KUKA KRL program: MyProgram_064().src

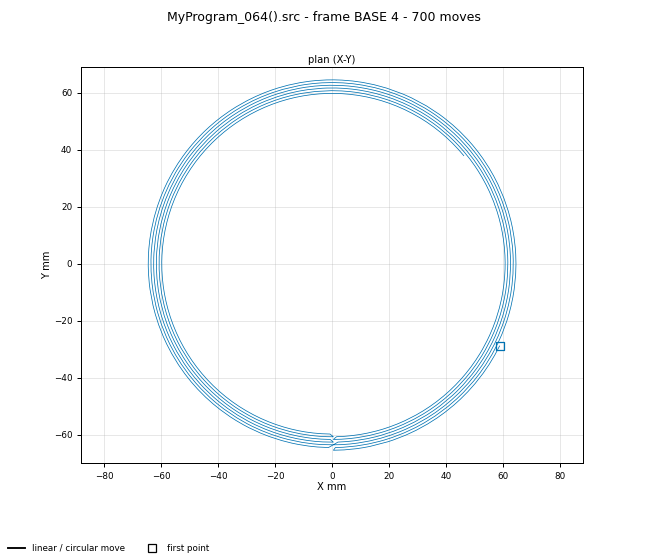
[picture p0: tool path of MyProgram_064().src in frame BASE 4, 700 of 700 moves have a stored position in this frame; points joined in program order, loops and branches not executed]
&ACCESS RVP
&REL 1
&PARAM TEMPLATE = C:\KRC\Roboter\Template\vorgabe
&PARAM EDITMASK = *
DEF MyProgram_064()
; ---- Setting reference (Base) ----
$BASE = BASE_DATA[4]

; --------------------------
; ---- Setting tool (TCP) ----
$TOOL = TOOL_DATA[3]
; --------------------------

$VEL.CP = VEL_APROX_PRINT
Startdeposition()
$VEL.CP = VEL_PRINT
LIN {X 58.7468,Y -28.8662,Z 73,A -33.1433,B 24.8941,C -2.3753,E1 25.1418,E2 117.3384} C_DIS
LIN {X 57.128,Y -31.9497,Z 73,A -36.5438,B 24.8957,C -2.3576,E1 25.1372,E2 120.763} C_DIS
LIN {X 55.082,Y -35.3604,Z 73,A -38.4998,B 24.8931,C -2.3868,E1 25.1344,E2 122.6401} C_DIS
LIN {X 52.9744,Y -38.4471,Z 73,A -42.3446,B 24.8952,C -2.3631,E1 25.1282,E2 126.522} C_DIS
LIN {X 50.1872,Y -42.0184,Z 73,A -46.4103,B 24.8964,C -2.3503,E1 25.1211,E2 130.5991} C_DIS
LIN {X 47.6348,Y -44.8923,Z 73,A -49.7399,B 24.897,C -2.3428,E1 25.1148,E2 133.9318} C_DIS
LIN {X 44.9577,Y -47.5733,Z 73,A -52.5816,B 24.8967,C -2.3469,E1 25.1092,E2 136.7518} C_DIS
LIN {X 42.7353,Y -49.5785,Z 73,A -55.4715,B 24.8978,C -2.3342,E1 25.1031,E2 139.6603} C_DIS
LIN {X 39.675,Y -52.0599,Z 73,A -59.4462,B 24.8996,C -2.3137,E1 25.0943,E2 143.6687} C_DIS
LIN {X 36.8552,Y -54.0936,Z 73,A -62.9268,B 24.901,C -2.297,E1 25.0862,E2 147.1772} C_DIS
LIN {X 33.4783,Y -56.2461,Z 73,A -64.9571,B 24.8984,C -2.3268,E1 25.0815,E2 149.1305} C_DIS
LIN {X 29.5121,Y -58.4253,Z 73,A -69.386,B 24.9,C -2.3085,E1 25.0706,E2 153.5901} C_DIS
LIN {X 25.8118,Y -60.1522,Z 73,A -72.5953,B 24.8997,C -2.3119,E1 25.0625,E2 156.7831} C_DIS
LIN {X 21.4205,Y -61.8516,Z 73,A -76.9276,B 24.9006,C -2.3013,E1 25.0511,E2 161.1313} C_DIS
LIN {X 19.5492,Y -62.468,Z 73,A -79.1991,B 24.9019,C -2.2862,E1 25.045,E2 163.4345} C_DIS
LIN {X 13.289,Y -64.0922,Z 73,A -83.8581,B 24.9004,C -2.3046,E1 25.0325,E2 168.0431} C_DIS
LIN {X 10.9976,Y -64.5247,Z 73,A -86.2924,B 24.9013,C -2.2936,E1 25.0257,E2 170.5007} C_DIS
LIN {X 8.6432,Y -64.8825,Z 73,A -88.6806,B 24.902,C -2.2851,E1 25.0191,E2 172.9071} C_DIS
LIN {X 4.2204,Y -65.3193,Z 73,A -92.8829,B 24.9028,C -2.2759,E1 25.0073,E2 177.1288} C_DIS
LIN {X 0.4624,Y -65.4389,Z 73,A -95.428,B 24.9014,C -2.2924,E1 25.0003,E2 179.6343} C_DIS
Enddeposition()
LIN {X 0.4624,Y -65.4389,Z 73,A -95.428,B 24.9014,C -2.2924,E1 25.0003,E2 179.6343} C_DIS
Startdeposition()
$VEL.CP = VEL_PRINT
LIN {X 1.1563,Y -64.495,Z 73,A -93.473,B 24.8973,C -2.3399,E1 25.0061,E2 177.5667} C_DIS
LIN {X 3.9215,Y -64.387,Z 73,A -91.3651,B 24.8979,C -2.3327,E1 25.0119,E2 175.4769} C_DIS
LIN {X 8.4282,Y -63.9525,Z 73,A -87.3099,B 24.8976,C -2.3358,E1 25.0232,E2 171.4172} C_DIS
LIN {X 12.7281,Y -63.2376,Z 73,A -83.9125,B 24.8984,C -2.3275,E1 25.0325,E2 168.0431} C_DIS
LIN {X 16.6215,Y -62.3274,Z 73,A -80.4027,B 24.8982,C -2.3299,E1 25.042,E2 164.5326} C_DIS
LIN {X 18.4457,Y -61.8118,Z 73,A -78.1953,B 24.8969,C -2.3443,E1 25.048,E2 162.2946} C_DIS
LIN {X 21.0877,Y -60.9617,Z 73,A -75.1268,B 24.8953,C -2.3621,E1 25.0562,E2 159.1901} C_DIS
LIN {X 25.2751,Y -59.3478,Z 73,A -71.5296,B 24.8957,C -2.3581,E1 25.0655,E2 155.6106} C_DIS
LIN {X 29.3295,Y -57.4519,Z 73,A -67.1057,B 24.8941,C -2.3757,E1 25.0766,E2 151.157} C_DIS
LIN {X 32.259,Y -55.8598,Z 73,A -65.0308,B 24.8956,C -2.3588,E1 25.0815,E2 149.1282} C_DIS
LIN {X 36.0916,Y -53.4634,Z 73,A -60.9163,B 24.8947,C -2.3688,E1 25.0912,E2 145.0033} C_DIS
LIN {X 40.6403,Y -50.093,Z 73,A -55.6203,B 24.8932,C -2.3861,E1 25.103,E2 139.6857} C_DIS
LIN {X 43.7386,Y -47.4121,Z 73,A -52.4535,B 24.8935,C -2.3824,E1 25.1096,E2 136.5403} C_DIS
LIN {X 46.088,Y -45.1316,Z 73,A -48.8099,B 24.8912,C -2.4081,E1 25.1169,E2 132.8512} C_DIS
LIN {X 49.6452,Y -41.1861,Z 73,A -44.3491,B 24.8907,C -2.4135,E1 25.125,E2 128.398} C_DIS
LIN {X 51.7521,Y -38.5064,Z 73,A -40.8175,B 24.8888,C -2.4346,E1 25.131,E2 124.8333} C_DIS
LIN {X 53.8109,Y -35.5715,Z 73,A -38.7033,B 24.8905,C -2.4156,E1 25.1342,E2 122.7745} C_DIS
LIN {X 56.1541,Y -31.7454,Z 73,A -34.9176,B 24.8899,C -2.4217,E1 25.1396,E2 118.9938} C_DIS
LIN {X 58.1359,Y -27.949,Z 73,A -31.0519,B 24.8888,C -2.4344,E1 25.1446,E2 115.1186} C_DIS
LIN {X 59.5801,Y -24.7239,Z 73,A -27.7511,B 24.8875,C -2.4479,E1 25.1483,E2 111.8037} C_DIS
LIN {X 61.2868,Y -20.1226,Z 73,A -23.7571,B 24.8872,C -2.4517,E1 25.1521,E2 107.8231} C_DIS
LIN {X 62.0906,Y -17.4843,Z 73,A -20.6908,B 24.885,C -2.4754,E1 25.1545,E2 104.7185} C_DIS
LIN {X 62.7454,Y -14.9688,Z 73,A -17.8709,B 24.8831,C -2.496,E1 25.1564,E2 101.8661} C_DIS
LIN {X 63.4244,Y -11.762,Z 73,A -15.9567,B 24.8847,C -2.479,E1 25.1573,E2 100.0033} C_DIS
LIN {X 63.8772,Y -8.9808,Z 73,A -12.9667,B 24.8827,C -2.4997,E1 25.1586,E2 96.982} C_DIS
LIN {X 64.3886,Y -3.8939,Z 73,A -8.1546,B 24.8807,C -2.5212,E1 25.1597,E2 92.1478} C_DIS
LIN {X 64.5052,Y -0.0652,Z 73,A -4.5358,B 24.8791,C -2.5377,E1 25.1597,E2 88.5115} C_DIS
LIN {X 64.4157,Y 3.4022,Z 73,A -2.7198,B 24.8813,C -2.5142,E1 25.1595,E2 86.7617} C_DIS
LIN {X 64.2639,Y 5.5868,Z 73,A -0.0027,B 24.8788,C -2.5404,E1 25.1589,E2 83.9987} C_DIS
LIN {X 63.8203,Y 9.3812,Z 73,A 3.0196,B 24.8788,C -2.5413,E1 25.1578,E2 80.9922} C_DIS
LIN {X 63.2661,Y 12.5892,Z 73,A 5.7276,B 24.8784,C -2.5454,E1 25.1564,E2 78.2903} C_DIS
LIN {X 62.7327,Y 15.0207,Z 73,A 8.8882,B 24.8753,C -2.5769,E1 25.1544,E2 75.0737} C_DIS
LIN {X 61.8474,Y 18.326,Z 73,A 11.5961,B 24.8753,C -2.5773,E1 25.1522,E2 72.3804} C_DIS
LIN {X 60.2454,Y 23.0538,Z 73,A 15.908,B 24.8744,C -2.5869,E1 25.1481,E2 68.0698} C_DIS
LIN {X 58.1702,Y 27.8777,Z 73,A 19.5732,B 24.8756,C -2.5744,E1 25.1441,E2 64.4542} C_DIS
LIN {X 56.6801,Y 30.7946,Z 73,A 23.2418,B 24.8729,C -2.6016,E1 25.1393,E2 60.7406} C_DIS
LIN {X 55.1029,Y 33.5352,Z 73,A 25.9438,B 24.8725,C -2.6062,E1 25.1354,E2 58.0416} C_DIS
LIN {X 52.9089,Y 36.8998,Z 73,A 29.262,B 24.8722,C -2.6088,E1 25.1303,E2 54.7336} C_DIS
LIN {X 51.0307,Y 39.4563,Z 73,A 32.2683,B 24.8711,C -2.6204,E1 25.1252,E2 51.7143} C_DIS
LIN {X 49.2652,Y 41.6406,Z 73,A 34.9272,B 24.8701,C -2.6302,E1 25.1204,E2 49.0442} C_DIS
LIN {X 47.4786,Y 43.666,Z 73,A 37.4243,B 24.8693,C -2.638,E1 25.1157,E2 46.5399} C_DIS
LIN {X 44.7609,Y 46.4478,Z 73,A 41.2384,B 24.8677,C -2.6541,E1 25.108,E2 42.7035} C_DIS
LIN {X 42.3154,Y 48.6864,Z 73,A 42.8652,B 24.8704,C -2.6272,E1 25.1048,E2 41.147} C_DIS
LIN {X 39.4678,Y 51.022,Z 73,A 46.1417,B 24.8698,C -2.6333,E1 25.0977,E2 37.8684} C_DIS
LIN {X 37.6241,Y 52.3966,Z 73,A 49.0641,B 24.8673,C -2.6583,E1 25.091,E2 34.8972} C_DIS
LIN {X 33.1232,Y 55.3526,Z 73,A 54.1357,B 24.8659,C -2.6725,E1 25.079,E2 29.8081} C_DIS
LIN {X 27.7921,Y 58.2114,Z 73,A 58.8294,B 24.8668,C -2.6629,E1 25.0674,E2 25.15} C_DIS
LIN {X 24.9466,Y 59.486,Z 73,A 62.2777,B 24.8649,C -2.6821,E1 25.0584,E2 21.6645} C_DIS
LIN {X 19.1378,Y 61.601,Z 73,A 67.412,B 24.8653,C -2.6781,E1 25.0449,E2 16.5496} C_DIS
LIN {X 14.7147,Y 62.8049,Z 73,A 71.1148,B 24.8659,C -2.672,E1 25.035,E2 12.8672} C_DIS
LIN {X 10.6426,Y 63.6213,Z 73,A 74.7482,B 24.8659,C -2.6721,E1 25.025,E2 9.2375} C_DIS
LIN {X 7.1714,Y 64.1051,Z 73,A 78.0569,B 24.8654,C -2.6772,E1 25.0158,E2 5.9193} C_DIS
LIN {X 3.4827,Y 64.4113,Z 73,A 81.5905,B 24.8648,C -2.6829,E1 25.0059,E2 2.3739} C_DIS
LIN {X 0.7153,Y 64.5022,Z 73,A 83.698,B 24.8657,C -2.6746,E1 25.0001,E2 0.2864} C_DIS
LIN {X -1.9461,Y 64.476,Z 73,A 86.182,B 24.8655,C -2.6766,E1 24.9932,E2 -2.2028} C_DIS
LIN {X -5.6035,Y 64.2621,Z 73,A 89.1745,B 24.8662,C -2.6695,E1 24.9849,E2 -5.1793} C_DIS
LIN {X -7.8512,Y 64.0265,Z 73,A 91.6622,B 24.8652,C -2.6789,E1 24.9779,E2 -7.6912} C_DIS
LIN {X -11.169,Y 63.5315,Z 73,A 93.8899,B 24.8671,C -2.6604,E1 24.9719,E2 -9.8769} C_DIS
LIN {X -15.3244,Y 62.6586,Z 73,A 97.4252,B 24.8679,C -2.6521,E1 24.9623,E2 -13.3967} C_DIS
LIN {X -18.975,Y 61.6515,Z 73,A 101.1903,B 24.8674,C -2.6572,E1 24.9521,E2 -17.1798} C_DIS
LIN {X -21.3436,Y 60.8719,Z 73,A 103.7868,B 24.8669,C -2.6626,E1 24.9452,E2 -19.7943} C_DIS
LIN {X -23.8319,Y 59.9421,Z 73,A 105.8647,B 24.8678,C -2.6535,E1 24.9398,E2 -21.8549} C_DIS
LIN {X -26.8305,Y 58.6604,Z 73,A 109.1217,B 24.8674,C -2.6569,E1 24.9314,E2 -25.1278} C_DIS
LIN {X -29.8299,Y 57.1928,Z 73,A 112.1913,B 24.8677,C -2.6544,E1 24.9238,E2 -28.1996} C_DIS
LIN {X -33.6214,Y 55.0505,Z 73,A 116.1114,B 24.8683,C -2.6486,E1 24.9144,E2 -32.1176} C_DIS
LIN {X -35.7625,Y 53.6849,Z 73,A 118.4897,B 24.8685,C -2.6468,E1 24.9088,E2 -34.4995} C_DIS
LIN {X -38.7189,Y 51.5925,Z 73,A 121.1599,B 24.8702,C -2.6291,E1 24.9029,E2 -37.1368} C_DIS
LIN {X -40.7762,Y 49.9828,Z 73,A 123.624,B 24.8704,C -2.6271,E1 24.8975,E2 -39.6053} C_DIS
LIN {X -43.021,Y 48.0638,Z 73,A 126.3383,B 24.8708,C -2.6231,E1 24.8918,E2 -42.3208} C_DIS
LIN {X -44.9132,Y 46.301,Z 73,A 128.3455,B 24.8719,C -2.6119,E1 24.8878,E2 -44.3096} C_DIS
LIN {X -47.0355,Y 44.143,Z 73,A 131.0757,B 24.8725,C -2.6062,E1 24.8825,E2 -47.0381} C_DIS
LIN {X -49.1146,Y 41.8173,Z 73,A 134.0295,B 24.8728,C -2.603,E1 24.877,E2 -49.9973} C_DIS
LIN {X -50.8555,Y 39.682,Z 73,A 136.4233,B 24.8735,C -2.5956,E1 24.8729,E2 -52.3846} C_DIS
LIN {X -52.3173,Y 37.7353,Z 73,A 139.0436,B 24.8732,C -2.5989,E1 24.8685,E2 -55.0256} C_DIS
LIN {X -54.1138,Y 35.1103,Z 73,A 141.9232,B 24.8738,C -2.5922,E1 24.8641,E2 -57.9037} C_DIS
LIN {X -56.0657,Y 31.9007,Z 73,A 145.8862,B 24.8735,C -2.5953,E1 24.8585,E2 -61.8947} C_DIS
LIN {X -57.8264,Y 28.584,Z 73,A 147.8932,B 24.877,C -2.5593,E1 24.8561,E2 -63.8264} C_DIS
LIN {X -58.8491,Y 26.4142,Z 73,A 150.8405,B 24.8761,C -2.569,E1 24.8526,E2 -66.8131} C_DIS
LIN {X -60.0746,Y 23.4945,Z 73,A 153.3783,B 24.8774,C -2.5551,E1 24.85,E2 -69.3319} C_DIS
LIN {X -61.2817,Y 20.139,Z 73,A 156.0607,B 24.8793,C -2.536,E1 24.8476,E2 -71.9838} C_DIS
LIN {X -62.395,Y 16.3677,Z 73,A 159.7267,B 24.88,C -2.5285,E1 24.8448,E2 -75.6532} C_DIS
LIN {X -63.4409,Y 11.673,Z 73,A 164.467,B 24.8804,C -2.5242,E1 24.842,E2 -80.4111} C_DIS
LIN {X -63.9424,Y 8.506,Z 73,A 167.1894,B 24.8815,C -2.5128,E1 24.8409,E2 -83.1225} C_DIS
LIN {X -64.2894,Y 5.2748,Z 73,A 169.9321,B 24.8826,C -2.5009,E1 24.8402,E2 -85.8531} C_DIS
LIN {X -64.4537,Y 2.5868,Z 73,A 172.7814,B 24.8825,C -2.5022,E1 24.8398,E2 -88.7227} C_DIS
LIN {X -64.5026,Y -0.6904,Z 73,A 175.1299,B 24.8844,C -2.482,E1 24.8398,E2 -91.0371} C_DIS
LIN {X -64.4131,Y -3.4495,Z 73,A 177.9855,B 24.8844,C -2.4822,E1 24.8402,E2 -93.9102} C_DIS
LIN {X -64.1273,Y -6.9783,Z 73,A -179.2847,B 24.886,C -2.4642,E1 24.8408,E2 -96.6136} C_DIS
LIN {X -63.8745,Y -8.9997,Z 73,A -177.1157,B 24.8859,C -2.4657,E1 24.8417,E2 -98.7989} C_DIS
LIN {X -62.8104,Y -14.6909,Z 73,A -172.4745,B 24.8883,C -2.4401,E1 24.8441,E2 -103.4064} C_DIS
LIN {X -61.9956,Y -17.8198,Z 73,A -168.0907,B 24.8863,C -2.4614,E1 24.8475,E2 -107.8666} C_DIS
LIN {X -60.8295,Y -21.4645,Z 73,A -165.918,B 24.8895,C -2.427,E1 24.8494,E2 -109.9696} C_DIS
LIN {X -59.2781,Y -25.4398,Z 73,A -161.8551,B 24.8899,C -2.4216,E1 24.8536,E2 -114.0421} C_DIS
LIN {X -58.0145,Y -28.2019,Z 73,A -158.1558,B 24.8888,C -2.4344,E1 24.8581,E2 -117.792} C_DIS
LIN {X -56.2629,Y -31.5505,Z 73,A -155.8796,B 24.8916,C -2.4035,E1 24.8611,E2 -120.0065} C_DIS
LIN {X -53.8835,Y -35.4614,Z 73,A -152.2506,B 24.8933,C -2.3842,E1 24.8664,E2 -123.6081} C_DIS
LIN {X -51.6586,Y -38.6308,Z 73,A -148.4743,B 24.8935,C -2.3826,E1 24.8725,E2 -127.3988} C_DIS
LIN {X -49.5171,Y -41.3402,Z 73,A -144.8664,B 24.8931,C -2.3865,E1 24.8789,E2 -131.033} C_DIS
LIN {X -47.1087,Y -44.0652,Z 73,A -141.5659,B 24.8936,C -2.3809,E1 24.8851,E2 -134.3347} C_DIS
LIN {X -44.345,Y -46.8455,Z 73,A -138.75,B 24.8955,C -2.3599,E1 24.8906,E2 -137.1124} C_DIS
LIN {X -41.6698,Y -49.2404,Z 73,A -135.7027,B 24.8963,C -2.3508,E1 24.897,E2 -140.15} C_DIS
LIN {X -39.2021,Y -51.2263,Z 73,A -132.6426,B 24.8963,C -2.3508,E1 24.9037,E2 -143.2217} C_DIS
LIN {X -35.7236,Y -53.7106,Z 73,A -128.9483,B 24.897,C -2.3424,E1 24.9121,E2 -146.9086} C_DIS
LIN {X -33.6688,Y -55.0217,Z 73,A -126.382,B 24.8966,C -2.3477,E1 24.9182,E2 -149.4957} C_DIS
LIN {X -31.0087,Y -56.5632,Z 73,A -123.8018,B 24.8972,C -2.3408,E1 24.9245,E2 -152.0669} C_DIS
LIN {X -29.1203,Y -57.5588,Z 73,A -121.5169,B 24.8967,C -2.3468,E1 24.9302,E2 -154.3723} C_DIS
LIN {X -25.066,Y -59.436,Z 73,A -117.0106,B 24.896,C -2.3545,E1 24.9418,E2 -158.9076} C_DIS
LIN {X -22.0591,Y -60.6163,Z 73,A -114.5932,B 24.8971,C -2.3419,E1 24.9481,E2 -161.3} C_DIS
LIN {X -17.6643,Y -62.0396,Z 73,A -110.5991,B 24.8976,C -2.3365,E1 24.9587,E2 -165.2882} C_DIS
LIN {X -14.1336,Y -62.9391,Z 73,A -107.5975,B 24.8982,C -2.3296,E1 24.9668,E2 -168.2773} C_DIS
LIN {X -11.91,Y -63.3958,Z 73,A -104.5581,B 24.8962,C -2.3522,E1 24.9753,E2 -171.3737} C_DIS
LIN {X -8.2112,Y -63.9806,Z 73,A -102.147,B 24.8981,C -2.3305,E1 24.9819,E2 -173.7351} C_DIS
LIN {X -5.2225,Y -64.2936,Z 73,A -99.2022,B 24.8976,C -2.3367,E1 24.9901,E2 -176.696} C_DIS
LIN {X -1.2767,Y -64.4928,Z 73,A -95.5948,B 24.8973,C -2.3394,E1 25.0002,E2 -180.3105} C_DIS
LIN {X -1.2767,Y -64.4928,Z 73,A -95.5948,B 24.8973,C -2.3394,E1 25.0002,E2 -180.3105} C_DIS
Enddeposition()
LIN {X 0.4502,Y -63.526,Z 73,A -94.7693,B 24.8973,C -2.3401,E1 25.0025,E2 -181.1376} C_DIS
Startdeposition()
$VEL.CP = VEL_PRINT
LIN {X -3.7985,Y -63.4425,Z 73,A -99.6016,B 24.8993,C -2.3166,E1 24.9888,E2 -176.2488} C_DIS
LIN {X -6.7271,Y -63.1985,Z 73,A -102.2235,B 24.8993,C -2.3174,E1 24.9815,E2 -173.6275} C_DIS
LIN {X -10.6276,Y -62.6607,Z 73,A -106.2689,B 24.9001,C -2.3076,E1 24.9703,E2 -169.5551} C_DIS
LIN {X -15.5509,Y -61.6242,Z 73,A -110.2262,B 24.8988,C -2.3222,E1 24.9596,E2 -165.6275} C_DIS
LIN {X -17.8908,Y -60.9853,Z 73,A -112.694,B 24.8992,C -2.3176,E1 24.9529,E2 -163.1449} C_DIS
LIN {X -21.2948,Y -59.8823,Z 73,A -116.714,B 24.9004,C -2.3036,E1 24.9422,E2 -159.0836} C_DIS
LIN {X -24.7528,Y -58.5371,Z 73,A -118.827,B 24.8979,C -2.3326,E1 24.937,E2 -157.0351} C_DIS
LIN {X -27.9356,Y -57.0876,Z 73,A -122.2592,B 24.8981,C -2.3303,E1 24.9282,E2 -153.5889} C_DIS
LIN {X -29.8114,Y -56.1304,Z 73,A -124.2589,B 24.8981,C -2.3307,E1 24.9233,E2 -151.5843} C_DIS
LIN {X -33.4,Y -54.0725,Z 73,A -128.1266,B 24.8979,C -2.3331,E1 24.914,E2 -147.7107} C_DIS
LIN {X -37.9663,Y -50.9698,Z 73,A -132.4905,B 24.8961,C -2.3537,E1 24.904,E2 -143.381} C_DIS
LIN {X -40.6133,Y -48.8861,Z 73,A -135.4758,B 24.8955,C -2.3601,E1 24.8975,E2 -140.4002} C_DIS
LIN {X -42.7747,Y -47.0067,Z 73,A -138.4364,B 24.8957,C -2.3575,E1 24.8913,E2 -137.4215} C_DIS
LIN {X -45.9463,Y -43.9124,Z 73,A -142.262,B 24.8947,C -2.3691,E1 24.8837,E2 -133.6074} C_DIS
LIN {X -47.8059,Y -41.8796,Z 73,A -145.1896,B 24.895,C -2.3658,E1 24.8782,E2 -130.6589} C_DIS
LIN {X -50.2885,Y -38.8635,Z 73,A -148.4282,B 24.8937,C -2.3795,E1 24.8726,E2 -127.4379} C_DIS
LIN {X -52.8793,Y -35.2587,Z 73,A -152.507,B 24.893,C -2.3878,E1 24.866,E2 -123.359} C_DIS
LIN {X -54.9846,Y -31.8755,Z 73,A -156.0304,B 24.892,C -2.3985,E1 24.8609,E2 -119.8429} C_DIS
LIN {X -56.8065,Y -28.5003,Z 73,A -159.7696,B 24.8917,C -2.4024,E1 24.856,E2 -116.0932} C_DIS
LIN {X -58.1144,Y -25.7321,Z 73,A -162.3869,B 24.8908,C -2.4128,E1 24.853,E2 -113.4863} C_DIS
LIN {X -59.8691,Y -21.3326,Z 73,A -166.725,B 24.8898,C -2.4237,E1 24.8486,E2 -109.15} C_DIS
LIN {X -61.2709,Y -16.8902,Z 73,A -171.0555,B 24.8888,C -2.4337,E1 24.8451,E2 -104.8184} C_DIS
LIN {X -61.7704,Y -14.9572,Z 73,A -173.4635,B 24.8894,C -2.4278,E1 24.8435,E2 -102.3821} C_DIS
LIN {X -62.7382,Y -10.163,Z 73,A -177.4879,B 24.8875,C -2.4484,E1 24.8415,E2 -98.3834} C_DIS
LIN {X -63.195,Y -6.7605,Z 73,A 179.7094,B 24.8861,C -2.4635,E1 24.8405,E2 -95.6} C_DIS
LIN {X -63.4977,Y -2.7039,Z 73,A 175.8031,B 24.8854,C -2.4706,E1 24.8399,E2 -91.687} C_DIS
LIN {X -63.5426,Y 1.2841,Z 73,A 172.2845,B 24.8842,C -2.4834,E1 24.8399,E2 -88.1778} C_DIS
LIN {X -63.4473,Y 3.7097,Z 73,A 170.3781,B 24.8831,C -2.4955,E1 24.8401,E2 -86.289} C_DIS
LIN {X -63.2082,Y 6.6348,Z 73,A 167.1731,B 24.8833,C -2.4935,E1 24.8409,E2 -83.0599} C_DIS
LIN {X -62.8176,Y 9.6561,Z 73,A 164.8611,B 24.8817,C -2.5103,E1 24.8418,E2 -80.7741} C_DIS
LIN {X -62.4549,Y 11.7785,Z 73,A 162.8495,B 24.8813,C -2.515,E1 24.8428,E2 -78.7621} C_DIS
LIN {X -61.624,Y 15.5515,Z 73,A 159.5903,B 24.8798,C -2.5301,E1 24.8448,E2 -75.5197} C_DIS
LIN {X -60.4183,Y 19.7217,Z 73,A 154.7618,B 24.8803,C -2.5251,E1 24.8488,E2 -70.6515} C_DIS
LIN {X -58.8753,Y 23.9373,Z 73,A 150.0331,B 24.8803,C -2.5248,E1 24.8537,E2 -65.8955} C_DIS
LIN {X -57.1956,Y 27.7128,Z 73,A 147.753,B 24.8767,C -2.5626,E1 24.8563,E2 -63.6934} C_DIS
LIN {X -54.973,Y 31.8957,Z 73,A 143.4451,B 24.8756,C -2.5741,E1 24.862,E2 -59.3902} C_DIS
LIN {X -53.9031,Y 33.6712,Z 73,A 140.8478,B 24.8764,C -2.5656,E1 24.8658,E2 -56.7593} C_DIS
LIN {X -51.6543,Y 37.029,Z 73,A 137.545,B 24.8748,C -2.5819,E1 24.871,E2 -53.4791} C_DIS
LIN {X -49.8108,Y 39.4738,Z 73,A 135.0334,B 24.8737,C -2.5939,E1 24.8753,E2 -50.9843} C_DIS
LIN {X -48.454,Y 41.1281,Z 73,A 132.3496,B 24.8746,C -2.5844,E1 24.8802,E2 -48.2655} C_DIS
LIN {X -44.9681,Y 44.9142,Z 73,A 128.2243,B 24.8725,C -2.6055,E1 24.888,E2 -44.1726} C_DIS
LIN {X -43.0497,Y 46.7549,Z 73,A 125.9285,B 24.8718,C -2.613,E1 24.8927,E2 -41.8853} C_DIS
LIN {X -41.1909,Y 48.4004,Z 73,A 123.729,B 24.8712,C -2.6187,E1 24.8973,E2 -39.6908} C_DIS
LIN {X -39.4304,Y 49.8451,Z 73,A 121.4963,B 24.8712,C -2.6196,E1 24.9022,E2 -37.4519} C_DIS
LIN {X -37.1121,Y 51.595,Z 73,A 118.6635,B 24.871,C -2.6207,E1 24.9086,E2 -34.6116} C_DIS
LIN {X -34.0821,Y 53.6451,Z 73,A 115.5229,B 24.8701,C -2.6301,E1 24.9159,E2 -31.4831} C_DIS
LIN {X -31.4466,Y 55.2311,Z 73,A 112.4741,B 24.8701,C -2.6295,E1 24.9233,E2 -28.4237} C_DIS
LIN {X -27.9052,Y 57.1027,Z 73,A 109.1629,B 24.869,C -2.6413,E1 24.9314,E2 -25.1317} C_DIS
LIN {X -24.7861,Y 58.5231,Z 73,A 106.1589,B 24.8684,C -2.6475,E1 24.9391,E2 -22.1354} C_DIS
LIN {X -21.0077,Y 59.9831,Z 73,A 102.3305,B 24.8683,C -2.6486,E1 24.9491,E2 -18.3018} C_DIS
LIN {X -17.264,Y 61.1658,Z 73,A 98.5447,B 24.8683,C -2.6475,E1 24.9593,E2 -14.5068} C_DIS
LIN {X -11.2802,Y 62.5464,Z 73,A 93.8654,B 24.8661,C -2.6702,E1 24.9719,E2 -9.8757} C_DIS
LIN {X -9.3924,Y 62.8576,Z 73,A 91.5957,B 24.8671,C -2.6599,E1 24.9782,E2 -7.5794} C_DIS
LIN {X -6.4948,Y 63.2228,Z 73,A 88.8376,B 24.8673,C -2.6587,E1 24.9859,E2 -4.8167} C_DIS
LIN {X -3.5543,Y 63.456,Z 73,A 86.2786,B 24.8669,C -2.6619,E1 24.993,E2 -2.2644} C_DIS
LIN {X 0.1727,Y 63.5556,Z 73,A 82.8264,B 24.8671,C -2.6608,E1 25.0026,E2 1.1907} C_DIS
LIN {X 3.8336,Y 63.4394,Z 73,A 79.4792,B 24.8671,C -2.66,E1 25.012,E2 4.5388} C_DIS
LIN {X 7.4768,Y 63.1142,Z 73,A 75.8987,B 24.8678,C -2.6534,E1 25.0219,E2 8.1326} C_DIS
LIN {X 10.6917,Y 62.65,Z 73,A 72.9261,B 24.868,C -2.6514,E1 25.0301,E2 11.1068} C_DIS
LIN {X 14.9359,Y 61.7756,Z 73,A 69.3195,B 24.8675,C -2.6562,E1 25.0399,E2 14.6974} C_DIS
LIN {X 18.3372,Y 60.8532,Z 73,A 65.3416,B 24.8695,C -2.6361,E1 25.0507,E2 18.7161} C_DIS
LIN {X 21.7721,Y 59.7099,Z 73,A 63.0845,B 24.8675,C -2.6559,E1 25.0565,E2 20.9216} C_DIS
LIN {X 25.2997,Y 58.3029,Z 73,A 59.5839,B 24.8681,C -2.6506,E1 25.0655,E2 24.4266} C_DIS
LIN {X 27.9916,Y 57.0599,Z 73,A 56.4298,B 24.8695,C -2.6364,E1 25.0735,E2 27.6061} C_DIS
LIN {X 32.6289,Y 54.5414,Z 73,A 52.5017,B 24.8682,C -2.6491,E1 25.083,E2 31.4926} C_DIS
LIN {X 34.4548,Y 53.4058,Z 73,A 50.395,B 24.8689,C -2.6422,E1 25.088,E2 33.6088} C_DIS
LIN {X 36.2153,Y 52.2279,Z 73,A 47.9023,B 24.8706,C -2.6255,E1 25.0938,E2 36.1328} C_DIS
LIN {X 38.8111,Y 50.3288,Z 73,A 44.8216,B 24.8715,C -2.6161,E1 25.1007,E2 39.2243} C_DIS
LIN {X 41.5761,Y 48.0709,Z 73,A 42.3802,B 24.8703,C -2.6284,E1 25.1058,E2 41.6272} C_DIS
LIN {X 44.281,Y 45.5911,Z 73,A 39.2645,B 24.8705,C -2.6264,E1 25.1122,E2 44.735} C_DIS
LIN {X 46.1792,Y 43.667,Z 73,A 36.8142,B 24.871,C -2.6209,E1 25.1169,E2 47.1879} C_DIS
LIN {X 48.1461,Y 41.4894,Z 73,A 33.8897,B 24.8723,C -2.6082,E1 25.1224,E2 50.1292} C_DIS
LIN {X 50.8543,Y 38.1199,Z 73,A 30.2544,B 24.8726,C -2.6054,E1 25.1287,E2 53.7541} C_DIS
LIN {X 51.8988,Y 36.6863,Z 73,A 28.0406,B 24.8744,C -2.5865,E1 25.1323,E2 56.0019} C_DIS
LIN {X 53.6234,Y 34.1158,Z 73,A 25.3869,B 24.8748,C -2.5827,E1 25.1363,E2 58.6512} C_DIS
LIN {X 55.5762,Y 30.832,Z 73,A 21.9153,B 24.8757,C -2.5729,E1 25.1411,E2 62.1279} C_DIS
LIN {X 57.3051,Y 27.4849,Z 73,A 18.8513,B 24.8758,C -2.5718,E1 25.1449,E2 65.1782} C_DIS
LIN {X 58.6645,Y 24.4506,Z 73,A 15.7975,B 24.8768,C -2.562,E1 25.1483,E2 68.2386} C_DIS
LIN {X 59.6866,Y 21.8358,Z 73,A 13.2718,B 24.8775,C -2.5548,E1 25.1508,E2 70.7672} C_DIS
LIN {X 60.9388,Y 18.0486,Z 73,A 9.2871,B 24.8794,C -2.5345,E1 25.1541,E2 74.7772} C_DIS
LIN {X 62.0005,Y 13.9764,Z 73,A 5.9868,B 24.8794,C -2.5353,E1 25.1563,E2 78.0565} C_DIS
LIN {X 62.4593,Y 11.7555,Z 73,A 3.5095,B 24.881,C -2.5182,E1 25.1576,E2 80.5597} C_DIS
LIN {X 63.2567,Y 6.1636,Z 73,A -1.0585,B 24.8812,C -2.5156,E1 25.1592,E2 85.107} C_DIS
LIN {X 63.4777,Y 3.1605,Z 73,A -3.4571,B 24.8812,C -2.515,E1 25.1596,E2 87.4927} C_DIS
LIN {X 63.5471,Y 1.0372,Z 73,A -6.0153,B 24.8834,C -2.4927,E1 25.1598,E2 90.0883} C_DIS
LIN {X 63.4584,Y -3.5105,Z 73,A -10.1636,B 24.8847,C -2.4786,E1 25.1593,E2 94.2454} C_DIS
LIN {X 63.1171,Y -7.4519,Z 73,A -12.9543,B 24.8839,C -2.4868,E1 25.1586,E2 97.0001} C_DIS
LIN {X 62.6944,Y -10.4262,Z 73,A -15.9996,B 24.8855,C -2.4697,E1 25.1573,E2 100.0679} C_DIS
LIN {X 61.8578,Y -14.5942,Z 73,A -19.467,B 24.8858,C -2.4669,E1 25.1553,E2 103.5216} C_DIS
LIN {X 60.8142,Y -18.4642,Z 73,A -23.165,B 24.887,C -2.4536,E1 25.1526,E2 107.23} C_DIS
LIN {X 59.7748,Y -21.5939,Z 73,A -26.6361,B 24.889,C -2.4319,E1 25.1494,E2 110.7328} C_DIS
LIN {X 58.2783,Y -25.3561,Z 73,A -30.2044,B 24.8898,C -2.423,E1 25.1455,E2 114.3025} C_DIS
LIN {X 56.9616,Y -28.19,Z 73,A -33.405,B 24.8914,C -2.4052,E1 25.1416,E2 117.5281} C_DIS
LIN {X 55.1771,Y -31.5405,Z 73,A -36.6365,B 24.8919,C -2.4001,E1 25.1372,E2 120.7549} C_DIS
LIN {X 52.8104,Y -35.3616,Z 73,A -40.4728,B 24.8924,C -2.3941,E1 25.1314,E2 124.5859} C_DIS
LIN {X 50.6371,Y -38.4092,Z 73,A -43.2733,B 24.892,C -2.3993,E1 25.1268,E2 127.3606} C_DIS
LIN {X 47.704,Y -41.9963,Z 73,A -47.508,B 24.8931,C -2.3871,E1 25.1192,E2 131.6047} C_DIS
LIN {X 44.6903,Y -45.1893,Z 73,A -51.6309,B 24.8943,C -2.3734,E1 25.1112,E2 135.7422} C_DIS
LIN {X 41.8553,Y -47.8271,Z 73,A -55.2572,B 24.8953,C -2.3621,E1 25.1037,E2 139.3807} C_DIS
LIN {X 39.376,Y -49.8881,Z 73,A -58.3644,B 24.8963,C -2.351,E1 25.0969,E2 142.5026} C_DIS
LIN {X 36.2374,Y -52.2125,Z 73,A -61.4801,B 24.8961,C -2.3536,E1 25.0898,E2 145.6011} C_DIS
LIN {X 33.2,Y -54.1951,Z 73,A -64.9224,B 24.897,C -2.3433,E1 25.0817,E2 149.0567} C_DIS
LIN {X 29.1469,Y -56.4784,Z 73,A -69.5424,B 24.8985,C -2.3261,E1 25.0703,E2 153.7043} C_DIS
LIN {X 25.7804,Y -58.0929,Z 73,A -71.9706,B 24.897,C -2.343,E1 25.0642,E2 156.0863} C_DIS
LIN {X 23.6332,Y -58.9991,Z 73,A -74.4555,B 24.898,C -2.331,E1 25.0578,E2 158.5939} C_DIS
LIN {X 20.5995,Y -60.1253,Z 73,A -76.9418,B 24.8975,C -2.3374,E1 25.0513,E2 161.0599} C_DIS
LIN {X 17.1264,Y -61.2048,Z 73,A -80.4569,B 24.8983,C -2.3281,E1 25.0419,E2 164.5908} C_DIS
LIN {X 13.123,Y -62.1868,Z 73,A -83.9196,B 24.8981,C -2.3304,E1 25.0325,E2 168.0431} C_DIS
LIN {X 9.0549,Y -62.9072,Z 73,A -87.7091,B 24.8985,C -2.3261,E1 25.022,E2 171.8389} C_DIS
LIN {X 6.267,Y -63.2467,Z 73,A -90.5312,B 24.8992,C -2.318,E1 25.0141,E2 174.6782} C_DIS
LIN {X 3.1859,Y -63.4763,Z 73,A -92.9305,B 24.8985,C -2.3255,E1 25.0075,E2 177.0586} C_DIS
LIN {X 0.4502,Y -63.526,Z 73,A -94.7678,B 24.8973,C -2.3395,E1 25.0025,E2 178.8624} C_DIS
Enddeposition()
LIN {X 0.4502,Y -63.526,Z 73,A -94.7678,B 24.8973,C -2.3395,E1 25.0025,E2 178.8624} C_DIS
Startdeposition()
$VEL.CP = VEL_PRINT
LIN {X 2.061,Y -62.5717,Z 73,A -93.0646,B 24.8954,C -2.361,E1 25.0074,E2 177.1086} C_DIS
LIN {X 4.9929,Y -62.4061,Z 73,A -90.3173,B 24.8952,C -2.3635,E1 25.015,E2 174.3564} C_DIS
LIN {X 7.8759,Y -62.1084,Z 73,A -87.2936,B 24.8943,C -2.3736,E1 25.0235,E2 171.311} C_DIS
LIN {X 12.3002,Y -61.386,Z 73,A -83.9199,B 24.8955,C -2.36,E1 25.0327,E2 167.9733} C_DIS
LIN {X 15.2208,Y -60.7278,Z 73,A -81.0528,B 24.895,C -2.3655,E1 25.0405,E2 165.0971} C_DIS
LIN {X 17.0774,Y -60.2313,Z 73,A -78.3756,B 24.8929,C -2.389,E1 25.0478,E2 162.3688} C_DIS
LIN {X 21.4718,Y -58.8083,Z 73,A -73.9616,B 24.892,C -2.3988,E1 25.0595,E2 157.9405} C_DIS
LIN {X 24.8575,Y -57.4594,Z 73,A -71.7882,B 24.8941,C -2.3758,E1 25.0649,E2 155.8265} C_DIS
LIN {X 28.8047,Y -55.5866,Z 73,A -67.9832,B 24.8939,C -2.3775,E1 25.0745,E2 152.0275} C_DIS
LIN {X 33.2455,Y -53.049,Z 73,A -62.9756,B 24.8925,C -2.3937,E1 25.0866,E2 146.9968} C_DIS
LIN {X 35.5688,Y -51.5204,Z 73,A -60.4254,B 24.892,C -2.3988,E1 25.0925,E2 144.4431} C_DIS
LIN {X 37.8986,Y -49.8326,Z 73,A -57.263,B 24.8903,C -2.4172,E1 25.0996,E2 141.2484} C_DIS
LIN {X 42.2396,Y -46.2091,Z 73,A -53.1535,B 24.8917,C -2.4026,E1 25.1083,E2 137.1896} C_DIS
LIN {X 43.6602,Y -44.8701,Z 73,A -50.8372,B 24.8901,C -2.4198,E1 25.113,E2 134.8423} C_DIS
LIN {X 45.8816,Y -42.5965,Z 73,A -47.685,B 24.8889,C -2.4329,E1 25.1191,E2 131.6726} C_DIS
LIN {X 49.1391,Y -38.7917,Z 73,A -43.3925,B 24.8885,C -2.4375,E1 25.1267,E2 127.3891} C_DIS
LIN {X 50.9341,Y -36.4029,Z 73,A -40.6493,B 24.8878,C -2.445,E1 25.1313,E2 124.6412} C_DIS
LIN {X 53.1724,Y -33.048,Z 73,A -36.7785,B 24.8864,C -2.4598,E1 25.1372,E2 120.7549} C_DIS
LIN {X 54.6546,Y -30.5339,Z 73,A -33.9575,B 24.8854,C -2.4712,E1 25.1411,E2 117.9216} C_DIS
LIN {X 56.17,Y -27.6481,Z 73,A -31.6776,B 24.8862,C -2.4622,E1 25.1439,E2 115.6751} C_DIS
LIN {X 57.2327,Y -25.3744,Z 73,A -28.8171,B 24.8843,C -2.4833,E1 25.1472,E2 112.7803} C_DIS
LIN {X 58.9458,Y -21.0919,Z 73,A -24.7019,B 24.8833,C -2.4934,E1 25.1513,E2 108.6642} C_DIS
LIN {X 59.8399,Y -18.4026,Z 73,A -22.5564,B 24.8836,C -2.49,E1 25.1531,E2 106.5389} C_DIS
LIN {X 60.7554,Y -15.1101,Z 73,A -19.4397,B 24.8827,C -2.4994,E1 25.1554,E2 103.4177} C_DIS
LIN {X 61.4116,Y -12.1705,Z 73,A -16.1884,B 24.8807,C -2.5207,E1 25.1573,E2 100.1352} C_DIS
LIN {X 61.9161,Y -9.2702,Z 73,A -13.8514,B 24.8807,C -2.5201,E1 25.1583,E2 97.8134} C_DIS
LIN {X 62.2628,Y -6.5414,Z 73,A -11.3058,B 24.88,C -2.5288,E1 25.1591,E2 95.2623} C_DIS
LIN {X 62.5909,Y -1.3707,Z 73,A -6.0127,B 24.8772,C -2.5578,E1 25.1598,E2 89.9319} C_DIS
LIN {X 62.5572,Y 2.4686,Z 73,A -3.163,B 24.8777,C -2.552,E1 25.1596,E2 87.1129} C_DIS
LIN {X 62.3783,Y 5.3411,Z 73,A -0.5123,B 24.8769,C -2.5607,E1 25.159,E2 84.4575} C_DIS
LIN {X 61.9601,Y 8.9679,Z 73,A 3.0327,B 24.8754,C -2.5762,E1 25.1578,E2 80.8966} C_DIS
LIN {X 61.4826,Y 11.8042,Z 73,A 5.3201,B 24.8754,C -2.5756,E1 25.1566,E2 78.6241} C_DIS
LIN {X 60.9474,Y 14.3151,Z 73,A 7.7658,B 24.8745,C -2.5852,E1 25.1551,E2 76.17} C_DIS
LIN {X 60.0303,Y 17.7712,Z 73,A 11.0458,B 24.8736,C -2.5951,E1 25.1527,E2 72.8852} C_DIS
LIN {X 59.3343,Y 19.9722,Z 73,A 13.7,B 24.8716,C -2.615,E1 25.1503,E2 70.1991} C_DIS
LIN {X 58.0357,Y 23.4803,Z 73,A 16.2868,B 24.8727,C -2.6038,E1 25.1477,E2 67.6531} C_DIS
LIN {X 56.5892,Y 26.7815,Z 73,A 19.8104,B 24.8713,C -2.6186,E1 25.1436,E2 64.1137} C_DIS
LIN {X 55.2045,Y 29.5304,Z 73,A 23.2362,B 24.869,C -2.6414,E1 25.1391,E2 60.652} C_DIS
LIN {X 52.9367,Y 33.4252,Z 73,A 26.3935,B 24.8703,C -2.6282,E1 25.1346,E2 57.5422} C_DIS
LIN {X 50.8848,Y 36.4719,Z 73,A 29.4895,B 24.8701,C -2.6301,E1 25.1298,E2 54.457} C_DIS
LIN {X 48.5754,Y 39.4955,Z 73,A 33.2243,B 24.8687,C -2.6445,E1 25.1234,E2 50.7057} C_DIS
LIN {X 47.0648,Y 41.2841,Z 73,A 35.7127,B 24.8674,C -2.6577,E1 25.1188,E2 48.1973} C_DIS
LIN {X 44.4334,Y 44.1038,Z 73,A 38.8678,B 24.8675,C -2.6562,E1 25.1128,E2 45.0593} C_DIS
LIN {X 42.7642,Y 45.7241,Z 73,A 41.686,B 24.8654,C -2.6771,E1 25.107,E2 42.2032} C_DIS
LIN {X 39.9129,Y 48.2331,Z 73,A 45.0683,B 24.865,C -2.6815,E1 25.0998,E2 38.8238} C_DIS
LIN {X 37.247,Y 50.3211,Z 73,A 48.2784,B 24.8642,C -2.6895,E1 25.0926,E2 35.6062} C_DIS
LIN {X 34.9373,Y 51.9507,Z 73,A 50.811,B 24.8639,C -2.6923,E1 25.0868,E2 33.0754} C_DIS
LIN {X 31.7832,Y 53.9378,Z 73,A 54.7704,B 24.8621,C -2.7102,E1 25.0772,E2 29.0857} C_DIS
LIN {X 28.523,Y 55.7305,Z 73,A 56.5836,B 24.8654,C -2.6775,E1 25.0729,E2 27.3554} C_DIS
LIN {X 26.8237,Y 56.5689,Z 73,A 58.9518,B 24.8637,C -2.6942,E1 25.0669,E2 24.9539} C_DIS
LIN {X 24.1623,Y 57.7552,Z 73,A 62.1631,B 24.8621,C -2.7096,E1 25.0586,E2 21.7135} C_DIS
LIN {X 20.9397,Y 59.0002,Z 73,A 65.6478,B 24.8611,C -2.7198,E1 25.0494,E2 18.2117} C_DIS
LIN {X 17.5321,Y 60.1012,Z 73,A 67.9341,B 24.8631,C -2.6995,E1 25.0434,E2 15.9776} C_DIS
LIN {X 15.1577,Y 60.7432,Z 73,A 70.5683,B 24.8621,C -2.7095,E1 25.0362,E2 13.3237} C_DIS
LIN {X 12.1169,Y 61.4221,Z 73,A 73.2143,B 24.8625,C -2.7062,E1 25.029,E2 10.6889} C_DIS
LIN {X 8.9488,Y 61.9628,Z 73,A 76.1285,B 24.8625,C -2.7064,E1 25.021,E2 7.7769} C_DIS
LIN {X 5.7892,Y 62.3373,Z 73,A 78.912,B 24.8627,C -2.704,E1 25.0133,E2 5.0011} C_DIS
LIN {X 2.8909,Y 62.5387,Z 73,A 81.6791,B 24.8624,C -2.7063,E1 25.0055,E2 2.2294} C_DIS
LIN {X -0.8046,Y 62.6004,Z 73,A 85.0122,B 24.8626,C -2.7046,E1 24.9962,E2 -1.0994} C_DIS
LIN {X -3.3249,Y 62.5173,Z 73,A 87.0548,B 24.8633,C -2.6982,E1 24.9906,E2 -3.1271} C_DIS
LIN {X -6.2665,Y 62.2916,Z 73,A 90.2635,B 24.8623,C -2.7078,E1 24.9816,E2 -6.3602} C_DIS
LIN {X -9.2494,Y 61.9191,Z 73,A 92.6056,B 24.8634,C -2.6974,E1 24.9752,E2 -8.6793} C_DIS
LIN {X -11.4148,Y 61.557,Z 73,A 94.6743,B 24.8634,C -2.6971,E1 24.9695,E2 -10.7496} C_DIS
LIN {X -15.0533,Y 60.7692,Z 73,A 98.167,B 24.8635,C -2.6959,E1 24.96,E2 -14.2438} C_DIS
LIN {X -18.9067,Y 59.6835,Z 73,A 101.559,B 24.8645,C -2.6863,E1 24.9509,E2 -17.6186} C_DIS
LIN {X -21.497,Y 58.7991,Z 73,A 104.6439,B 24.8636,C -2.6952,E1 24.9427,E2 -20.7307} C_DIS
LIN {X -23.927,Y 57.8539,Z 73,A 106.7686,B 24.8645,C -2.6865,E1 24.9373,E2 -22.8394} C_DIS
LIN {X -26.6689,Y 56.6418,Z 73,A 109.4185,B 24.8651,C -2.6805,E1 24.9306,E2 -25.4816} C_DIS
LIN {X -28.9492,Y 55.51,Z 73,A 112.4269,B 24.8641,C -2.6906,E1 24.923,E2 -28.5221} C_DIS
LIN {X -32.6686,Y 53.4064,Z 73,A 116.5679,B 24.8643,C -2.6882,E1 24.9131,E2 -32.6702} C_DIS
LIN {X -35.4065,Y 51.6325,Z 73,A 118.7194,B 24.8666,C -2.6657,E1 24.9082,E2 -34.7752} C_DIS
LIN {X -37.8738,Y 49.8512,Z 73,A 121.7382,B 24.8666,C -2.6647,E1 24.9014,E2 -37.8022} C_DIS
LIN {X -40.5173,Y 47.7264,Z 73,A 124.8575,B 24.8673,C -2.6583,E1 24.8947,E2 -40.9181} C_DIS
LIN {X -43.1109,Y 45.3981,Z 73,A 127.9956,B 24.8681,C -2.65,E1 24.8883,E2 -44.0491} C_DIS
LIN {X -45.5701,Y 42.9281,Z 73,A 131.1811,B 24.8689,C -2.6422,E1 24.8821,E2 -47.2298} C_DIS
LIN {X -47.7933,Y 40.4388,Z 73,A 134.2199,B 24.8697,C -2.6342,E1 24.8765,E2 -50.2633} C_DIS
LIN {X -49.8729,Y 37.8449,Z 73,A 137.4606,B 24.8701,C -2.6301,E1 24.871,E2 -53.5094} C_DIS
LIN {X -51.5825,Y 35.4794,Z 73,A 140.1503,B 24.8708,C -2.6232,E1 24.8667,E2 -56.1959} C_DIS
LIN {X -53.6881,Y 32.2037,Z 73,A 143.1215,B 24.8729,C -2.602,E1 24.8623,E2 -59.1317} C_DIS
LIN {X -54.7013,Y 30.4504,Z 73,A 146.1035,B 24.8713,C -2.6183,E1 24.8582,E2 -62.1681} C_DIS
LIN {X -56.6649,Y 26.6187,Z 73,A 150.0819,B 24.8724,C -2.6074,E1 24.8534,E2 -66.1421} C_DIS
LIN {X -58.363,Y 22.6556,Z 73,A 153.3531,B 24.8748,C -2.5827,E1 24.85,E2 -69.3725} C_DIS
LIN {X -59.5553,Y 19.3034,Z 73,A 156.8388,B 24.8753,C -2.5771,E1 24.8468,E2 -72.8647} C_DIS
LIN {X -60.6502,Y 15.5243,Z 73,A 160.2678,B 24.8767,C -2.5627,E1 24.8443,E2 -76.2792} C_DIS
LIN {X -61.4424,Y 12.0133,Z 73,A 163.8016,B 24.8773,C -2.5569,E1 24.8423,E2 -79.8199} C_DIS
LIN {X -61.9703,Y 8.8961,Z 73,A 166.9467,B 24.8777,C -2.5525,E1 24.841,E2 -82.9733} C_DIS
LIN {X -62.491,Y 3.7937,Z 73,A 170.9254,B 24.8804,C -2.5242,E1 24.84,E2 -86.9082} C_DIS
LIN {X -62.5656,Y 2.2389,Z 73,A 172.7989,B 24.88,C -2.5281,E1 24.8398,E2 -88.8024} C_DIS
LIN {X -62.5947,Y -1.1626,Z 73,A 175.7025,B 24.8813,C -2.5144,E1 24.8398,E2 -91.6906} C_DIS
LIN {X -62.4833,Y -3.9222,Z 73,A 178.4945,B 24.8816,C -2.5114,E1 24.8403,E2 -94.4921} C_DIS
LIN {X -62.2627,Y -6.5427,Z 73,A -179.5457,B 24.8831,C -2.4955,E1 24.8408,E2 -96.4257} C_DIS
LIN {X -61.934,Y -9.1461,Z 73,A -176.9116,B 24.8834,C -2.4924,E1 24.8418,E2 -99.0682} C_DIS
LIN {X -61.4422,Y -12.0142,Z 73,A -174.0395,B 24.8838,C -2.4882,E1 24.8432,E2 -101.9473} C_DIS
LIN {X -60.7273,Y -15.2244,Z 73,A -171.4222,B 24.8853,C -2.4716,E1 24.8449,E2 -104.5403} C_DIS
LIN {X -59.9687,Y -17.9771,Z 73,A -168.4612,B 24.8854,C -2.4705,E1 24.8472,E2 -107.5156} C_DIS
LIN {X -58.9322,Y -21.132,Z 73,A -165.7779,B 24.8869,C -2.4548,E1 24.8495,E2 -110.1768} C_DIS
LIN {X -57.8283,Y -23.9888,Z 73,A -162.9472,B 24.8876,C -2.4473,E1 24.8524,E2 -113.0054} C_DIS
LIN {X -57.0139,Y -25.8629,Z 73,A -160.7801,B 24.8876,C -2.4477,E1 24.8549,E2 -115.1856} C_DIS
LIN {X -55.587,Y -28.8015,Z 73,A -157.4904,B 24.8878,C -2.4454,E1 24.859,E2 -118.4874} C_DIS
LIN {X -54.4374,Y -30.9212,Z 73,A -155.1391,B 24.888,C -2.4424,E1 24.8623,E2 -120.8437} C_DIS
LIN {X -51.8772,Y -35.0459,Z 73,A -151.6162,B 24.8907,C -2.4131,E1 24.8675,E2 -124.3146} C_DIS
LIN {X -50.2955,Y -37.282,Z 73,A -148.5572,B 24.8903,C -2.4178,E1 24.8725,E2 -127.3996} C_DIS
LIN {X -48.4122,Y -39.6966,Z 73,A -144.8329,B 24.8892,C -2.4296,E1 24.8791,E2 -131.1695} C_DIS
LIN {X -46.181,Y -42.2702,Z 73,A -143.1342,B 24.8924,C -2.3945,E1 24.8822,E2 -132.792} C_DIS
LIN {X -44.8608,Y -43.6699,Z 73,A -140.294,B 24.8908,C -2.4122,E1 24.8878,E2 -135.6868} C_DIS
LIN {X -41.682,Y -46.7126,Z 73,A -136.6398,B 24.8922,C -2.3967,E1 24.8952,E2 -139.3189} C_DIS
LIN {X -39.8673,Y -48.271,Z 73,A -134.1076,B 24.8919,C -2.3997,E1 24.9007,E2 -141.8677} C_DIS
LIN {X -36.6791,Y -50.7369,Z 73,A -130.2246,B 24.8921,C -2.3974,E1 24.9094,E2 -145.759} C_DIS
LIN {X -33.1306,Y -53.1207,Z 73,A -126.7385,B 24.8935,C -2.3826,E1 24.9176,E2 -149.2211} C_DIS
LIN {X -29.5619,Y -55.1874,Z 73,A -123.1361,B 24.8943,C -2.3739,E1 24.9263,E2 -152.8133} C_DIS
LIN {X -27.0142,Y -56.4774,Z 73,A -119.9511,B 24.8934,C -2.3829,E1 24.9344,E2 -156.0279} C_DIS
LIN {X -23.6529,Y -57.9655,Z 73,A -116.3259,B 24.8933,C -2.3851,E1 24.9438,E2 -159.6666} C_DIS
LIN {X -20.527,Y -59.1451,Z 73,A -114.1871,B 24.8952,C -2.3628,E1 24.9493,E2 -161.7565} C_DIS
LIN {X -18.1181,Y -59.9274,Z 73,A -111.7179,B 24.8952,C -2.3643,E1 24.9559,E2 -164.2337} C_DIS
LIN {X -15.2643,Y -60.7171,Z 73,A -108.4614,B 24.8942,C -2.3747,E1 24.9647,E2 -167.5195} C_DIS
LIN {X -12.2365,Y -61.3991,Z 73,A -105.2834,B 24.8936,C -2.381,E1 24.9735,E2 -170.7161} C_DIS
LIN {X -8.7633,Y -61.9892,Z 73,A -103.0186,B 24.8956,C -2.359,E1 24.9796,E2 -172.9305} C_DIS
LIN {X -6.0581,Y -62.3125,Z 73,A -100.5179,B 24.8956,C -2.3588,E1 24.9866,E2 -175.4324} C_DIS
LIN {X -3.2828,Y -62.5196,Z 73,A -97.5205,B 24.8947,C -2.369,E1 24.995,E2 -178.455} C_DIS
LIN {X 0.441,Y -62.5875,Z 73,A -95.0084,B 24.8964,C -2.3498,E1 25.0019,E2 -180.9216} C_DIS
Enddeposition()
LIN {X 0.441,Y -62.5875,Z 73,A -95.0084,B 24.8964,C -2.3498,E1 25.0019,E2 -180.9216} C_DIS
Startdeposition()
$VEL.CP = VEL_PRINT
LIN {X -0.6544,Y -61.6528,Z 73,A -97.0446,B 24.8969,C -2.3436,E1 24.9962,E2 -178.8706} C_DIS
LIN {X -3.8981,Y -61.5328,Z 73,A -99.9045,B 24.8967,C -2.3468,E1 24.9882,E2 -176.0174} C_DIS
LIN {X -6.8374,Y -61.2762,Z 73,A -102.5678,B 24.8965,C -2.3487,E1 24.9808,E2 -173.3572} C_DIS
LIN {X -9.0044,Y -60.9955,Z 73,A -105.1056,B 24.8974,C -2.3384,E1 24.9737,E2 -170.793} C_DIS
LIN {X -11.8012,Y -60.5159,Z 73,A -107.4388,B 24.8968,C -2.3457,E1 24.9674,E2 -168.4746} C_DIS
LIN {X -14.9777,Y -59.8099,Z 73,A -110.4171,B 24.8965,C -2.3482,E1 24.9593,E2 -165.4982} C_DIS
LIN {X -18.3468,Y -58.8627,Z 73,A -113.5751,B 24.8962,C -2.3524,E1 24.9508,E2 -162.3449} C_DIS
LIN {X -21.6643,Y -57.7244,Z 73,A -116.8801,B 24.896,C -2.3542,E1 24.9421,E2 -159.0377} C_DIS
LIN {X -24.311,Y -56.6614,Z 73,A -119.7308,B 24.8961,C -2.3528,E1 24.9348,E2 -156.1771} C_DIS
LIN {X -27.2809,Y -55.2918,Z 73,A -122.5345,B 24.8954,C -2.3611,E1 24.9277,E2 -153.386} C_DIS
LIN {X -29.3118,Y -54.2424,Z 73,A -125.3013,B 24.8963,C -2.3511,E1 24.9208,E2 -150.5876} C_DIS
LIN {X -32.8612,Y -52.169,Z 73,A -128.2291,B 24.8942,C -2.3742,E1 24.914,E2 -147.7058} C_DIS
LIN {X -35.0439,Y -50.7284,Z 73,A -130.9085,B 24.8943,C -2.3731,E1 24.9077,E2 -145.0149} C_DIS
LIN {X -37.4612,Y -48.9706,Z 73,A -133.9444,B 24.8943,C -2.3728,E1 24.9009,E2 -141.9675} C_DIS
LIN {X -39.6818,Y -47.19,Z 73,A -136.3083,B 24.8934,C -2.3831,E1 24.8958,E2 -139.6192} C_DIS
LIN {X -42.3611,Y -44.7994,Z 73,A -139.7453,B 24.893,C -2.3878,E1 24.8887,E2 -136.1794} C_DIS
LIN {X -44.4069,Y -42.7719,Z 73,A -142.4532,B 24.8926,C -2.3928,E1 24.8834,E2 -133.472} C_DIS
LIN {X -46.3614,Y -40.6454,Z 73,A -145.5057,B 24.8926,C -2.3917,E1 24.8777,E2 -130.4033} C_DIS
LIN {X -48.8262,Y -37.6486,Z 73,A -148.6607,B 24.8911,C -2.4086,E1 24.8723,E2 -127.2738} C_DIS
LIN {X -50.6356,Y -35.1774,Z 73,A -151.0378,B 24.8897,C -2.4244,E1 24.8684,E2 -124.9228} C_DIS
LIN {X -52.1112,Y -32.9521,Z 73,A -154.2923,B 24.8904,C -2.4162,E1 24.8634,E2 -121.6323} C_DIS
LIN {X -53.8244,Y -30.0723,Z 73,A -157.0682,B 24.8891,C -2.4306,E1 24.8596,E2 -118.8764} C_DIS
LIN {X -55.4281,Y -27.0047,Z 73,A -160.4293,B 24.8886,C -2.4367,E1 24.8553,E2 -115.5117} C_DIS
LIN {X -56.5595,Y -24.5448,Z 73,A -162.9809,B 24.888,C -2.4431,E1 24.8524,E2 -112.9615} C_DIS
LIN {X -57.7935,Y -21.4816,Z 73,A -165.7709,B 24.8867,C -2.4569,E1 24.8496,E2 -110.1889} C_DIS
LIN {X -58.8852,Y -18.2743,Z 73,A -169.931,B 24.8875,C -2.4479,E1 24.8459,E2 -105.9834} C_DIS
LIN {X -60.3136,Y -12.7889,Z 73,A -174.8414,B 24.8855,C -2.4702,E1 24.8428,E2 -101.0977} C_DIS
LIN {X -60.981,Y -9.0864,Z 73,A -178.4826,B 24.8847,C -2.4784,E1 24.8411,E2 -97.4543} C_DIS
LIN {X -61.4383,Y -5.1772,Z 73,A 177.9404,B 24.8835,C -2.4912,E1 24.8401,E2 -93.8866} C_DIS
LIN {X -61.6403,Y -1.3988,Z 73,A 174.521,B 24.8823,C -2.504,E1 24.8398,E2 -90.4772} C_DIS
LIN {X -61.6033,Y 2.542,Z 73,A 171.3521,B 24.8804,C -2.5245,E1 24.84,E2 -87.3381} C_DIS
LIN {X -61.5172,Y 4.1295,Z 73,A 169.0544,B 24.8813,C -2.5145,E1 24.8404,E2 -85.0026} C_DIS
LIN {X -60.9531,Y 9.2822,Z 73,A 164.1774,B 24.88,C -2.5286,E1 24.8421,E2 -80.1304} C_DIS
LIN {X -60.0506,Y 13.9768,Z 73,A 160.2179,B 24.8778,C -2.5512,E1 24.8444,E2 -76.2014} C_DIS
LIN {X -58.6923,Y 18.885,Z 73,A 155.3975,B 24.8766,C -2.5642,E1 24.8481,E2 -71.3842} C_DIS
LIN {X -57.7927,Y 21.4838,Z 73,A 152.8186,B 24.8759,C -2.5715,E1 24.8505,E2 -68.8082} C_DIS
LIN {X -56.9622,Y 23.5979,Z 73,A 150.4074,B 24.8758,C -2.5725,E1 24.8531,E2 -66.3859} C_DIS
LIN {X -55.6448,Y 26.5536,Z 73,A 147.8429,B 24.8741,C -2.5893,E1 24.8561,E2 -63.8477} C_DIS
LIN {X -53.7633,Y 30.1817,Z 73,A 143.8595,B 24.8734,C -2.5969,E1 24.8613,E2 -59.8613} C_DIS
LIN {X -52.0829,Y 32.9984,Z 73,A 140.2058,B 24.8736,C -2.5944,E1 24.8667,E2 -56.1829} C_DIS
LIN {X -50.3284,Y 35.6163,Z 73,A 137.5231,B 24.8724,C -2.6068,E1 24.871,E2 -53.5166} C_DIS
LIN {X -47.7097,Y 39.055,Z 73,A 134.0523,B 24.8704,C -2.6273,E1 24.8769,E2 -50.0784} C_DIS
LIN {X -46.4588,Y 40.5338,Z 73,A 131.3213,B 24.8716,C -2.6147,E1 24.882,E2 -47.3049} C_DIS
LIN {X -43.6391,Y 43.5563,Z 73,A 127.8657,B 24.87,C -2.631,E1 24.8886,E2 -43.8734} C_DIS
LIN {X -40.6907,Y 46.3211,Z 73,A 124.5336,B 24.8684,C -2.6475,E1 24.8954,E2 -40.5672} C_DIS
LIN {X -39.0594,Y 47.7061,Z 73,A 122.0831,B 24.8688,C -2.6431,E1 24.9008,E2 -38.0969} C_DIS
LIN {X -35.4811,Y 50.4245,Z 73,A 117.6887,B 24.8684,C -2.6474,E1 24.9107,E2 -33.6974} C_DIS
LIN {X -31.3511,Y 53.0898,Z 73,A 113.2621,B 24.8673,C -2.6585,E1 24.9212,E2 -29.2833} C_DIS
LIN {X -27.8653,Y 54.9999,Z 73,A 109.7158,B 24.8664,C -2.6674,E1 24.9299,E2 -25.7484} C_DIS
LIN {X -24.9427,Y 56.386,Z 73,A 106.8745,B 24.8656,C -2.6751,E1 24.9371,E2 -22.9184} C_DIS
LIN {X -23.2526,Y 57.1028,Z 73,A 104.5418,B 24.8666,C -2.6652,E1 24.9432,E2 -20.557} C_DIS
LIN {X -19.1371,Y 58.6107,Z 73,A 100.5459,B 24.866,C -2.6716,E1 24.9537,E2 -16.5687} C_DIS
LIN {X -14.9561,Y 59.8152,Z 73,A 97.0699,B 24.8644,C -2.687,E1 24.963,E2 -13.124} C_DIS
LIN {X -11.702,Y 60.535,Z 73,A 93.5976,B 24.8649,C -2.6821,E1 24.9725,E2 -9.6359} C_DIS
LIN {X -8.5279,Y 61.0632,Z 73,A 90.4444,B 24.8651,C -2.6807,E1 24.9813,E2 -6.4768} C_DIS
LIN {X -3.478,Y 61.5575,Z 73,A 86.421,B 24.8634,C -2.6971,E1 24.9924,E2 -2.4905} C_DIS
LIN {X -1.7981,Y 61.6295,Z 73,A 84.4902,B 24.8641,C -2.6899,E1 24.9978,E2 -0.5423} C_DIS
LIN {X 1.4749,Y 61.6389,Z 73,A 81.6236,B 24.8637,C -2.694,E1 25.0058,E2 2.3142} C_DIS
LIN {X 4.063,Y 61.5212,Z 73,A 78.9822,B 24.8642,C -2.6892,E1 25.0132,E2 4.9661} C_DIS
LIN {X 7.06,Y 61.2502,Z 73,A 76.5577,B 24.8634,C -2.6967,E1 25.0198,E2 7.3712} C_DIS
LIN {X 9.3702,Y 60.9394,Z 73,A 74.293,B 24.8637,C -2.694,E1 25.0261,E2 9.6402} C_DIS
LIN {X 12.5222,Y 60.3707,Z 73,A 71.3817,B 24.8637,C -2.6942,E1 25.0341,E2 12.5476} C_DIS
LIN {X 15.3804,Y 59.7064,Z 73,A 68.5351,B 24.8641,C -2.6901,E1 25.0418,E2 15.3999} C_DIS
LIN {X 18.7526,Y 58.7351,Z 73,A 65.2105,B 24.8645,C -2.6864,E1 25.0507,E2 18.7275} C_DIS
LIN {X 21.4008,Y 57.8231,Z 73,A 62.3256,B 24.8653,C -2.6779,E1 25.0583,E2 21.6266} C_DIS
LIN {X 24.7921,Y 56.4517,Z 73,A 59.2344,B 24.865,C -2.6812,E1 25.0662,E2 24.7029} C_DIS
LIN {X 27.5162,Y 55.1751,Z 73,A 56.4584,B 24.8653,C -2.6783,E1 25.0732,E2 27.4784} C_DIS
LIN {X 31.1139,Y 53.23,Z 73,A 52.7584,B 24.8656,C -2.6754,E1 25.0823,E2 31.1744} C_DIS
LIN {X 33.6176,Y 51.6856,Z 73,A 49.8986,B 24.8663,C -2.6683,E1 25.089,E2 34.0417} C_DIS
LIN {X 36.6379,Y 49.5898,Z 73,A 46.7018,B 24.8663,C -2.6677,E1 25.0963,E2 37.229} C_DIS
LIN {X 38.6864,Y 48.0084,Z 73,A 43.9136,B 24.8677,C -2.6545,E1 25.1024,E2 40.0379} C_DIS
LIN {X 42.5881,Y 44.5841,Z 73,A 39.6982,B 24.8672,C -2.6592,E1 25.1111,E2 44.2255} C_DIS
LIN {X 45.134,Y 42.0052,Z 73,A 35.9509,B 24.8688,C -2.6431,E1 25.1185,E2 47.9947} C_DIS
LIN {X 47.131,Y 39.7515,Z 73,A 33.2891,B 24.8691,C -2.64,E1 25.1233,E2 50.6518} C_DIS
LIN {X 49.6605,Y 36.5414,Z 73,A 29.4605,B 24.8701,C -2.6303,E1 25.1299,E2 54.4853} C_DIS
LIN {X 51.7606,Y 33.5009,Z 73,A 26.2395,B 24.8704,C -2.6267,E1 25.1349,E2 57.6988} C_DIS
LIN {X 52.799,Y 31.8391,Z 73,A 23.9253,B 24.8721,C -2.6103,E1 25.1383,E2 60.0401} C_DIS
LIN {X 54.472,Y 28.8834,Z 73,A 21.1464,B 24.8721,C -2.6108,E1 25.142,E2 62.8031} C_DIS
LIN {X 55.6928,Y 26.4538,Z 73,A 18.9097,B 24.8721,C -2.6108,E1 25.1447,E2 65.0277} C_DIS
LIN {X 57.4345,Y 22.4212,Z 73,A 13.7185,B 24.8757,C -2.5726,E1 25.1503,E2 70.2808} C_DIS
LIN {X 58.547,Y 19.3336,Z 73,A 11.6855,B 24.8742,C -2.5882,E1 25.1521,E2 72.2656} C_DIS
LIN {X 59.1218,Y 17.4938,Z 73,A 9.5784,B 24.8755,C -2.5752,E1 25.1538,E2 74.3913} C_DIS
LIN {X 59.9794,Y 14.2829,Z 73,A 6.6427,B 24.876,C -2.5696,E1 25.1559,E2 77.3233} C_DIS
LIN {X 60.5364,Y 11.6942,Z 73,A 4.1902,B 24.8767,C -2.5623,E1 25.1572,E2 79.7788} C_DIS
LIN {X 61.03,Y 8.7613,Z 73,A 1.2855,B 24.8779,C -2.5503,E1 25.1585,E2 82.6948} C_DIS
LIN {X 61.4183,Y 5.4103,Z 73,A -1.6392,B 24.8783,C -2.5457,E1 25.1593,E2 85.6131} C_DIS
LIN {X 61.5941,Y 2.7559,Z 73,A -4.1322,B 24.8791,C -2.5374,E1 25.1597,E2 88.1109} C_DIS
LIN {X 61.6537,Y 0.5331,Z 73,A -6.4423,B 24.8803,C -2.5249,E1 25.1597,E2 90.4368} C_DIS
LIN {X 61.5261,Y -3.9978,Z 73,A -10.3926,B 24.881,C -2.518,E1 25.1593,E2 94.38} C_DIS
LIN {X 61.2645,Y -6.9378,Z 73,A -12.9991,B 24.8815,C -2.5126,E1 25.1586,E2 96.9837} C_DIS
LIN {X 60.8805,Y -9.7514,Z 73,A -15.3942,B 24.8817,C -2.5103,E1 25.1576,E2 99.3702} C_DIS
LIN {X 60.4008,Y -12.3756,Z 73,A -18.1891,B 24.8832,C -2.4947,E1 25.1562,E2 102.1855} C_DIS
LIN {X 59.8256,Y -14.9132,Z 73,A -20.6743,B 24.884,C -2.4855,E1 25.1545,E2 104.6782} C_DIS
LIN {X 59.0297,Y -17.804,Z 73,A -23.2975,B 24.8845,C -2.4808,E1 25.1525,E2 107.2973} C_DIS
LIN {X 57.9098,Y -21.1629,Z 73,A -26.614,B 24.8855,C -2.4701,E1 25.1495,E2 110.6205} C_DIS
LIN {X 56.8316,Y -23.9079,Z 73,A -29.1364,B 24.8858,C -2.4672,E1 25.1468,E2 113.1358} C_DIS
LIN {X 55.6629,Y -26.516,Z 73,A -32.3957,B 24.8878,C -2.4447,E1 25.143,E2 116.4309} C_DIS
LIN {X 53.7679,Y -30.1736,Z 73,A -35.5892,B 24.8874,C -2.449,E1 25.1388,E2 119.5974} C_DIS
LIN {X 52.5341,Y -32.275,Z 73,A -38.3837,B 24.8892,C -2.4298,E1 25.1347,E2 122.423} C_DIS
LIN {X 50.4652,Y -35.4226,Z 73,A -41.5516,B 24.8893,C -2.4282,E1 25.1297,E2 125.579} C_DIS
LIN {X 48.6323,Y -37.9003,Z 73,A -44.2255,B 24.8896,C -2.4251,E1 25.1253,E2 128.2474} C_DIS
LIN {X 46.7644,Y -40.1818,Z 73,A -47.5228,B 24.8915,C -2.4048,E1 25.1193,E2 131.5777} C_DIS
LIN {X 44.0429,Y -43.1474,Z 73,A -50.7599,B 24.8912,C -2.4076,E1 25.1131,E2 134.794} C_DIS
LIN {X 41.9268,Y -45.2069,Z 73,A -53.443,B 24.8917,C -2.4026,E1 25.1077,E2 137.4779} C_DIS
LIN {X 39.4847,Y -47.3538,Z 73,A -56.7861,B 24.893,C -2.3883,E1 25.1005,E2 140.8418} C_DIS
LIN {X 36.6635,Y -49.5711,Z 73,A -59.8075,B 24.893,C -2.3886,E1 25.0938,E2 143.8514} C_DIS
LIN {X 34.4143,Y -51.1576,Z 73,A -62.3911,B 24.8934,C -2.383,E1 25.0879,E2 146.4396} C_DIS
LIN {X 31.9441,Y -52.7351,Z 73,A -65.3529,B 24.8944,C -2.3724,E1 25.0808,E2 149.4171} C_DIS
LIN {X 28.7808,Y -54.526,Z 73,A -68.8345,B 24.8951,C -2.3642,E1 25.0723,E2 152.9081} C_DIS
LIN {X 24.9363,Y -56.3889,Z 73,A -72.6158,B 24.8953,C -2.3624,E1 25.0627,E2 156.684} C_DIS
LIN {X 21.8585,Y -57.6509,Z 73,A -75.5363,B 24.8953,C -2.3621,E1 25.0551,E2 159.5988} C_DIS
LIN {X 19.0913,Y -58.6255,Z 73,A -78.0779,B 24.8953,C -2.3629,E1 25.0484,E2 162.1335} C_DIS
LIN {X 17.0285,Y -59.2579,Z 73,A -80.7407,B 24.8967,C -2.3459,E1 25.0412,E2 164.832} C_DIS
LIN {X 12.9567,Y -60.2791,Z 73,A -83.8388,B 24.8955,C -2.3601,E1 25.0329,E2 167.892} C_DIS
LIN {X 8.9688,Y -61.0005,Z 73,A -87.912,B 24.8963,C -2.3504,E1 25.0216,E2 171.984} C_DIS
LIN {X 6.1112,Y -61.3528,Z 73,A -90.5886,B 24.8965,C -2.3488,E1 25.0142,E2 174.6624} C_DIS
LIN {X 3.176,Y -61.5742,Z 73,A -93.2974,B 24.8965,C -2.3483,E1 25.0066,E2 177.3714} C_DIS
LIN {X 0.4357,Y -61.6466,Z 73,A -95.2691,B 24.8955,C -2.3602,E1 25.0012,E2 179.3145} C_DIS
Enddeposition()
LIN {X 0.4357,Y -61.6466,Z 73,A -95.2691,B 24.8955,C -2.3602,E1 25.0012,E2 179.3145} C_DIS
Startdeposition()
$VEL.CP = VEL_PRINT
LIN {X 1.5855,Y -60.6856,Z 73,A -93.5499,B 24.8928,C -2.3906,E1 25.0062,E2 177.5234} C_DIS
LIN {X 4.3801,Y -60.5482,Z 73,A -90.8332,B 24.8925,C -2.3933,E1 25.0138,E2 174.8013} C_DIS
LIN {X 7.1583,Y -60.2823,Z 73,A -88.2134,B 24.8925,C -2.3945,E1 25.0211,E2 172.1804} C_DIS
LIN {X 10.0813,Y -59.8628,Z 73,A -85.2957,B 24.892,C -2.3994,E1 25.0292,E2 169.2539} C_DIS
LIN {X 12.5067,Y -59.4042,Z 73,A -83.1373,B 24.8921,C -2.3976,E1 25.035,E2 167.1026} C_DIS
LIN {X 15.6457,Y -58.6552,Z 73,A -80.3987,B 24.8925,C -2.3937,E1 25.0424,E2 164.3772} C_DIS
LIN {X 17.7411,Y -58.056,Z 73,A -78.0326,B 24.8916,C -2.403,E1 25.0488,E2 161.9932} C_DIS
LIN {X 20.3649,Y -57.1886,Z 73,A -75.3861,B 24.8913,C -2.4071,E1 25.0558,E2 159.3422} C_DIS
LIN {X 23.0038,Y -56.1785,Z 73,A -72.8289,B 24.8912,C -2.4083,E1 25.0624,E2 156.7879} C_DIS
LIN {X 25.5512,Y -55.0666,Z 73,A -69.3804,B 24.8891,C -2.4314,E1 25.0713,E2 153.2933} C_DIS
LIN {X 29.5058,Y -53.0528,Z 73,A -66.1047,B 24.8904,C -2.4171,E1 25.0793,E2 150.0607} C_DIS
LIN {X 31.8614,Y -51.6736,Z 73,A -63.345,B 24.8895,C -2.4261,E1 25.0859,E2 147.2883} C_DIS
LIN {X 34.3942,Y -50.0232,Z 73,A -60.5574,B 24.8892,C -2.4301,E1 25.0924,E2 144.5006} C_DIS
LIN {X 36.7082,Y -48.3507,Z 73,A -57.8955,B 24.8887,C -2.4349,E1 25.0983,E2 141.8368} C_DIS
LIN {X 39.0373,Y -46.4905,Z 73,A -55.0622,B 24.8881,C -2.4415,E1 25.1045,E2 138.9986} C_DIS
LIN {X 41.245,Y -44.5433,Z 73,A -52.3064,B 24.8876,C -2.4473,E1 25.1102,E2 136.2401} C_DIS
LIN {X 43.3381,Y -42.5093,Z 73,A -49.5738,B 24.887,C -2.4534,E1 25.1156,E2 133.5048} C_DIS
LIN {X 45.2884,Y -40.4247,Z 73,A -46.8632,B 24.8864,C -2.4605,E1 25.1207,E2 130.7894} C_DIS
LIN {X 46.9375,Y -38.499,Z 73,A -44.5012,B 24.8859,C -2.4659,E1 25.1249,E2 128.4254} C_DIS
LIN {X 48.6759,Y -36.2753,Z 73,A -41.832,B 24.8852,C -2.4731,E1 25.1295,E2 125.7518} C_DIS
LIN {X 50.4092,Y -33.8255,Z 73,A -39.1267,B 24.8848,C -2.4777,E1 25.1337,E2 123.0489} C_DIS
LIN {X 51.8937,Y -31.4996,Z 73,A -36.8135,B 24.8848,C -2.478,E1 25.1372,E2 120.7468} C_DIS
LIN {X 52.6971,Y -30.1366,Z 73,A -35.0059,B 24.8836,C -2.4899,E1 25.1397,E2 118.9204} C_DIS
LIN {X 54.4231,Y -26.8946,Z 73,A -31.9051,B 24.8836,C -2.491,E1 25.1437,E2 115.8332} C_DIS
LIN {X 55.322,Y -24.9932,Z 73,A -29.5962,B 24.8822,C -2.5048,E1 25.1464,E2 113.5042} C_DIS
LIN {X 56.4543,Y -22.3185,Z 73,A -26.8617,B 24.8815,C -2.5129,E1 25.1493,E2 110.7658} C_DIS
LIN {X 57.4192,Y -19.706,Z 73,A -24.1724,B 24.8806,C -2.5224,E1 25.1518,E2 108.069} C_DIS
LIN {X 58.6872,Y -15.5266,Z 73,A -20.128,B 24.8795,C -2.5332,E1 25.155,E2 104.0221} C_DIS
LIN {X 59.3889,Y -12.5809,Z 73,A -17.4323,B 24.8791,C -2.5382,E1 25.1566,E2 101.3304} C_DIS
LIN {X 59.7573,Y -10.6891,Z 73,A -15.5138,B 24.8783,C -2.5464,E1 25.1576,E2 99.4038} C_DIS
LIN {X 60.2017,Y -7.8066,Z 73,A -12.7254,B 24.8774,C -2.556,E1 25.1587,E2 96.6091} C_DIS
LIN {X 60.5106,Y -4.8636,Z 73,A -10.0019,B 24.8767,C -2.5631,E1 25.1594,E2 93.885} C_DIS
LIN {X 60.674,Y -1.966,Z 73,A -7.2382,B 24.8758,C -2.5724,E1 25.1597,E2 91.1158} C_DIS
LIN {X 60.704,Y 0.4723,Z 73,A -5.1124,B 24.8755,C -2.5753,E1 25.1597,E2 88.9956} C_DIS
LIN {X 60.6331,Y 2.9895,Z 73,A -2.5898,B 24.8744,C -2.5864,E1 25.1595,E2 86.4619} C_DIS
LIN {X 60.4092,Y 6.0014,Z 73,A 0.1711,B 24.8738,C -2.5931,E1 25.1588,E2 83.7014} C_DIS
LIN {X 60.0999,Y 8.5547,Z 73,A 2.3639,B 24.8736,C -2.5949,E1 25.158,E2 81.5174} C_DIS
LIN {X 59.7359,Y 10.808,Z 73,A 4.6669,B 24.8726,C -2.6052,E1 25.1569,E2 79.2035} C_DIS
LIN {X 59.2364,Y 13.2798,Z 73,A 7.157,B 24.8716,C -2.6151,E1 25.1555,E2 76.7045} C_DIS
LIN {X 58.5491,Y 16.0385,Z 73,A 9.7048,B 24.8711,C -2.6199,E1 25.1537,E2 74.1601} C_DIS
LIN {X 57.8717,Y 18.3343,Z 73,A 12.3704,B 24.8695,C -2.6365,E1 25.1514,E2 71.4704} C_DIS
LIN {X 56.6652,Y 21.7791,Z 73,A 15.4808,B 24.8693,C -2.6383,E1 25.1485,E2 68.3731} C_DIS
LIN {X 55.2106,Y 25.2404,Z 73,A 18.9356,B 24.8685,C -2.6461,E1 25.1446,E2 64.9187} C_DIS
LIN {X 54.0252,Y 27.685,Z 73,A 21.5576,B 24.8677,C -2.6545,E1 25.1413,E2 62.2907} C_DIS
LIN {X 52.626,Y 30.2603,Z 73,A 24.3193,B 24.867,C -2.6618,E1 25.1376,E2 59.5263} C_DIS
LIN {X 51.2131,Y 32.5954,Z 73,A 26.8637,B 24.8664,C -2.6676,E1 25.1338,E2 56.9809} C_DIS
LIN {X 50.0295,Y 34.3851,Z 73,A 28.8246,B 24.866,C -2.6712,E1 25.1307,E2 55.0213} C_DIS
LIN {X 48.3507,Y 36.7082,Z 73,A 31.7601,B 24.8648,C -2.6832,E1 25.1258,E2 52.0715} C_DIS
LIN {X 46.2232,Y 39.3523,Z 73,A 34.7243,B 24.8646,C -2.6849,E1 25.1205,E2 49.1168} C_DIS
LIN {X 44.3325,Y 41.4709,Z 73,A 37.4103,B 24.864,C -2.6909,E1 25.1155,E2 46.4285} C_DIS
LIN {X 42.9516,Y 42.9005,Z 73,A 39.2816,B 24.8636,C -2.6947,E1 25.1118,E2 44.5561} C_DIS
LIN {X 40.8032,Y 44.9487,Z 73,A 42.0571,B 24.8631,C -2.6997,E1 25.1061,E2 41.78} C_DIS
LIN {X 37.446,Y 47.7812,Z 73,A 45.8698,B 24.8631,C -2.6997,E1 25.098,E2 37.9819} C_DIS
LIN {X 35.5268,Y 49.2254,Z 73,A 48.5064,B 24.8619,C -2.7121,E1 25.092,E2 35.3254} C_DIS
LIN {X 32.9672,Y 50.9744,Z 73,A 51.2612,B 24.8618,C -2.7128,E1 25.0856,E2 32.578} C_DIS
LIN {X 30.5277,Y 52.4724,Z 73,A 54.1334,B 24.861,C -2.7206,E1 25.0787,E2 29.6963} C_DIS
LIN {X 28.0607,Y 53.8316,Z 73,A 56.7174,B 24.8608,C -2.7224,E1 25.0723,E2 27.1153} C_DIS
LIN {X 25.2968,Y 55.185,Z 73,A 59.6164,B 24.8605,C -2.7257,E1 25.065,E2 24.2161} C_DIS
LIN {X 22.4693,Y 56.395,Z 73,A 62.4923,B 24.8602,C -2.7281,E1 25.0576,E2 21.3412} C_DIS
LIN {X 19.6144,Y 57.4501,Z 73,A 65.2729,B 24.8602,C -2.7286,E1 25.0503,E2 18.5652} C_DIS
LIN {X 16.3969,Y 58.4495,Z 73,A 68.4536,B 24.8599,C -2.7309,E1 25.0418,E2 15.3845} C_DIS
LIN {X 11.702,Y 59.5676,Z 73,A 72.8365,B 24.8601,C -2.7294,E1 25.0299,E2 11.0111} C_DIS
LIN {X 9.0342,Y 60.0302,Z 73,A 75.8224,B 24.859,C -2.7395,E1 25.0216,E2 8.0043} C_DIS
LIN {X 6.2157,Y 60.3868,Z 73,A 78.0859,B 24.8599,C -2.731,E1 25.0154,E2 5.7625} C_DIS
LIN {X 3.331,Y 60.6143,Z 73,A 81.134,B 24.8592,C -2.7378,E1 25.0068,E2 2.6996} C_DIS
LIN {X -0.2274,Y 60.7047,Z 73,A 84.9344,B 24.8583,C -2.7465,E1 24.9962,E2 -1.1212} C_DIS
LIN {X -5.8954,Y 60.4196,Z 73,A 90.4298,B 24.8583,C -2.7471,E1 24.9809,E2 -6.6202} C_DIS
LIN {X -10.8264,Y 59.7326,Z 73,A 94.6248,B 24.8597,C -2.7335,E1 24.9694,E2 -10.7865} C_DIS
LIN {X -14.6247,Y 58.9182,Z 73,A 97.8621,B 24.8609,C -2.7215,E1 24.9606,E2 -13.9996} C_DIS
LIN {X -17.5769,Y 58.105,Z 73,A 101.0131,B 24.8607,C -2.7237,E1 24.9521,E2 -17.1608} C_DIS
LIN {X -20.2725,Y 57.221,Z 73,A 103.7775,B 24.8608,C -2.7222,E1 24.9448,E2 -19.927} C_DIS
LIN {X -23.0594,Y 56.1559,Z 73,A 106.2922,B 24.8618,C -2.7125,E1 24.9383,E2 -22.4239} C_DIS
LIN {X -25.2408,Y 55.2104,Z 73,A 108.8666,B 24.8615,C -2.7157,E1 24.9317,E2 -25.0121} C_DIS
LIN {X -28.0136,Y 53.8565,Z 73,A 111.9808,B 24.8615,C -2.715,E1 24.924,E2 -28.133} C_DIS
LIN {X -30.2295,Y 52.6437,Z 73,A 114.0467,B 24.8626,C -2.7047,E1 24.919,E2 -30.1804} C_DIS
LIN {X -32.5665,Y 51.2316,Z 73,A 116.6611,B 24.863,C -2.7007,E1 24.9128,E2 -32.7935} C_DIS
LIN {X -35.0387,Y 49.5736,Z 73,A 120.0453,B 24.8625,C -2.7063,E1 24.905,E2 -36.2025} C_DIS
LIN {X -38.8723,Y 46.6276,Z 73,A 123.8347,B 24.8649,C -2.6819,E1 24.8968,E2 -39.9477} C_DIS
LIN {X -41.2898,Y 44.5022,Z 73,A 127.5919,B 24.8643,C -2.6886,E1 24.8889,E2 -43.7359} C_DIS
LIN {X -43.3311,Y 42.5163,Z 73,A 130.1999,B 24.8651,C -2.6806,E1 24.8838,E2 -46.336} C_DIS
LIN {X -46.2626,Y 39.306,Z 73,A 133.6355,B 24.8673,C -2.658,E1 24.8775,E2 -49.7329} C_DIS
LIN {X -48.5684,Y 36.4184,Z 73,A 137.551,B 24.8675,C -2.6568,E1 24.8707,E2 -53.664} C_DIS
LIN {X -50.0213,Y 34.3959,Z 73,A 140.6287,B 24.8667,C -2.6639,E1 24.8658,E2 -56.7739} C_DIS
LIN {X -52.3023,Y 30.8166,Z 73,A 143.827,B 24.8694,C -2.6378,E1 24.8612,E2 -59.9263} C_DIS
LIN {X -53.6504,Y 28.4048,Z 73,A 146.5356,B 24.8699,C -2.6322,E1 24.8576,E2 -62.6357} C_DIS
LIN {X -55.5876,Y 24.3973,Z 73,A 150.597,B 24.8714,C -2.6172,E1 24.8528,E2 -66.6836} C_DIS
LIN {X -56.5014,Y 22.1986,Z 73,A 153.0559,B 24.8717,C -2.6143,E1 24.8502,E2 -69.1492} C_DIS
LIN {X -57.435,Y 19.659,Z 73,A 155.5319,B 24.8726,C -2.6051,E1 24.8479,E2 -71.6173} C_DIS
LIN {X -58.3836,Y 16.6295,Z 73,A 158.5174,B 24.8735,C -2.5957,E1 24.8455,E2 -74.5975} C_DIS
LIN {X -59.0882,Y 13.9227,Z 73,A 161.2614,B 24.8741,C -2.5894,E1 24.8436,E2 -77.3424} C_DIS
LIN {X -60.0191,Y 9.106,Z 73,A 165.932,B 24.8755,C -2.5755,E1 24.8413,E2 -82.0075} C_DIS
LIN {X -60.5492,Y 4.3647,Z 73,A 170.0779,B 24.8775,C -2.5549,E1 24.8402,E2 -86.1288} C_DIS
LIN {X -60.6577,Y 2.4203,Z 73,A 173.04,B 24.8761,C -2.5694,E1 24.8398,E2 -89.1435} C_DIS
LIN {X -60.6753,Y -1.9206,Z 73,A 177.2332,B 24.8771,C -2.5582,E1 24.8401,E2 -93.3353} C_DIS
LIN {X -60.4493,Y -5.5741,Z 73,A 179.9789,B 24.8794,C -2.5345,E1 24.8407,E2 -96.0407} C_DIS
LIN {X -59.7985,Y -10.4598,Z 73,A -175.4539,B 24.8809,C -2.5185,E1 24.8425,E2 -100.5969} C_DIS
LIN {X -58.9048,Y -14.6798,Z 73,A -171.2233,B 24.8818,C -2.509,E1 24.8451,E2 -104.8298} C_DIS
LIN {X -58.0972,Y -17.6074,Z 73,A -167.5302,B 24.8812,C -2.5158,E1 24.8481,E2 -108.5603} C_DIS
LIN {X -57.0565,Y -20.7304,Z 73,A -165.7907,B 24.8844,C -2.4816,E1 24.8496,E2 -110.228} C_DIS
LIN {X -56.3711,Y -22.5304,Z 73,A -163.4336,B 24.884,C -2.4862,E1 24.852,E2 -112.6093} C_DIS
LIN {X -55.3761,Y -24.8733,Z 73,A -161.0476,B 24.8846,C -2.4792,E1 24.8547,E2 -114.9917} C_DIS
LIN {X -54.2405,Y -27.263,Z 73,A -158.0335,B 24.8844,C -2.482,E1 24.8584,E2 -118.0287} C_DIS
LIN {X -52.9822,Y -29.6322,Z 73,A -155.2478,B 24.8846,C -2.4801,E1 24.8623,E2 -120.8245} C_DIS
LIN {X -49.8356,Y -34.664,Z 73,A -150.2615,B 24.887,C -2.4542,E1 24.8698,E2 -125.7742} C_DIS
LIN {X -48.1999,Y -36.9052,Z 73,A -147.6787,B 24.8876,C -2.4473,E1 24.8741,E2 -128.3528} C_DIS
LIN {X -46.5476,Y -38.9686,Z 73,A -145.462,B 24.8886,C -2.4362,E1 24.878,E2 -130.5534} C_DIS
LIN {X -45.0051,Y -40.7412,Z 73,A -142.9295,B 24.8886,C -2.4373,E1 24.8827,E2 -133.0998} C_DIS
LIN {X -42.9809,Y -42.8709,Z 73,A -140.1147,B 24.889,C -2.4323,E1 24.8882,E2 -135.9147} C_DIS
LIN {X -40.8668,Y -44.8904,Z 73,A -137.1864,B 24.8892,C -2.4301,E1 24.8942,E2 -138.8497} C_DIS
LIN {X -38.7293,Y -46.7465,Z 73,A -134.6685,B 24.8899,C -2.4221,E1 24.8996,E2 -141.3583} C_DIS
LIN {X -36.4772,Y -48.5242,Z 73,A -131.9784,B 24.8904,C -2.417,E1 24.9055,E2 -144.046} C_DIS
LIN {X -34.2086,Y -50.1498,Z 73,A -129.3026,B 24.8907,C -2.4136,E1 24.9117,E2 -146.7227} C_DIS
LIN {X -32.1195,Y -51.5124,Z 73,A -126.03,B 24.8893,C -2.4285,E1 24.9195,E2 -150.0413} C_DIS
LIN {X -29.0617,Y -53.2974,Z 73,A -123.7508,B 24.8917,C -2.4025,E1 24.925,E2 -152.2651} C_DIS
LIN {X -26.6092,Y -54.5642,Z 73,A -121.0311,B 24.8917,C -2.4017,E1 24.9317,E2 -154.99} C_DIS
LIN {X -23.8439,Y -55.8278,Z 73,A -118.1788,B 24.8921,C -2.3982,E1 24.939,E2 -157.841} C_DIS
LIN {X -21.1717,Y -56.8952,Z 73,A -115.2647,B 24.8919,C -2.3998,E1 24.9466,E2 -160.765} C_DIS
LIN {X -18.793,Y -57.7236,Z 73,A -112.5584,B 24.8915,C -2.4048,E1 24.9539,E2 -163.4882} C_DIS
LIN {X -14.6908,Y -58.9021,Z 73,A -108.8404,B 24.8923,C -2.3959,E1 24.9639,E2 -167.1906} C_DIS
LIN {X -11.0147,Y -59.6987,Z 73,A -105.8411,B 24.8935,C -2.3828,E1 24.972,E2 -170.1623} C_DIS
LIN {X -7.3476,Y -60.2601,Z 73,A -102.0006,B 24.8929,C -2.3892,E1 24.9826,E2 -174.0212} C_DIS
LIN {X -4.5358,Y -60.5368,Z 73,A -99.315,B 24.8929,C -2.3895,E1 24.9901,E2 -176.7087} C_DIS
LIN {X -1.903,Y -60.6759,Z 73,A -96.7751,B 24.8927,C -2.3909,E1 24.9972,E2 -179.2524} C_DIS
LIN {X 0.4349,Y -60.7034,Z 73,A -95.5655,B 24.8946,C -2.3699,E1 25.0005,E2 -180.4121} C_DIS
Enddeposition()
LIN {X 0.4349,Y -60.7034,Z 73,A -95.5655,B 24.8946,C -2.3699,E1 25.0005,E2 -180.4121} C_DIS
Startdeposition()
$VEL.CP = VEL_PRINT
LIN {X -0.7426,Y -59.7523,Z 73,A -97.0497,B 24.8938,C -2.3787,E1 24.9964,E2 -178.949} C_DIS
LIN {X -3.669,Y -59.6442,Z 73,A -99.8572,B 24.8938,C -2.3785,E1 24.9885,E2 -176.1403} C_DIS
LIN {X -6.5868,Y -59.3928,Z 73,A -102.6668,B 24.8938,C -2.3787,E1 24.9807,E2 -173.3296} C_DIS
LIN {X -9.5006,Y -58.9968,Z 73,A -105.1524,B 24.8931,C -2.3862,E1 24.9739,E2 -170.8597} C_DIS
LIN {X -11.7946,Y -58.5807,Z 73,A -107.6114,B 24.8935,C -2.3825,E1 24.9671,E2 -168.3892} C_DIS
LIN {X -14.3275,Y -58.013,Z 73,A -110.1998,B 24.8935,C -2.3817,E1 24.9601,E2 -165.7955} C_DIS
LIN {X -16.9673,Y -57.2963,Z 73,A -112.832,B 24.8935,C -2.3832,E1 24.953,E2 -163.1627} C_DIS
LIN {X -19.7423,Y -56.4004,Z 73,A -115.6436,B 24.8932,C -2.3851,E1 24.9456,E2 -160.3504} C_DIS
LIN {X -22.1923,Y -55.4832,Z 73,A -118.1573,B 24.893,C -2.3873,E1 24.939,E2 -157.8366} C_DIS
LIN {X -24.8891,Y -54.327,Z 73,A -120.9788,B 24.8928,C -2.3902,E1 24.9318,E2 -155.0151} C_DIS
LIN {X -27.5204,Y -53.0426,Z 73,A -123.7955,B 24.8925,C -2.3934,E1 24.9248,E2 -152.1987} C_DIS
LIN {X -30.1346,Y -51.602,Z 73,A -126.6808,B 24.8922,C -2.3969,E1 24.9178,E2 -149.3131} C_DIS
LIN {X -32.624,Y -50.0653,Z 73,A -129.4563,B 24.8918,C -2.4017,E1 24.9112,E2 -146.5402} C_DIS
LIN {X -35.0076,Y -48.4289,Z 73,A -132.2626,B 24.8914,C -2.4056,E1 24.9048,E2 -143.7335} C_DIS
LIN {X -37.3417,Y -46.6529,Z 73,A -135.1021,B 24.891,C -2.41,E1 24.8986,E2 -140.8941} C_DIS
LIN {X -39.5967,Y -44.7547,Z 73,A -137.9237,B 24.8905,C -2.4154,E1 24.8926,E2 -138.0745} C_DIS
LIN {X -41.7381,Y -42.7647,Z 73,A -140.74,B 24.89,C -2.4209,E1 24.8869,E2 -135.2595} C_DIS
LIN {X -43.7802,Y -40.6716,Z 73,A -143.5596,B 24.8895,C -2.4265,E1 24.8815,E2 -132.4412} C_DIS
LIN {X -45.7174,Y -38.4813,Z 73,A -146.3778,B 24.8889,C -2.4326,E1 24.8763,E2 -129.6246} C_DIS
LIN {X -47.5568,Y -36.1834,Z 73,A -149.2207,B 24.8884,C -2.4388,E1 24.8715,E2 -126.7833} C_DIS
LIN {X -49.1704,Y -33.9568,Z 73,A -151.8035,B 24.8877,C -2.4463,E1 24.8673,E2 -124.2056} C_DIS
LIN {X -50.7336,Y -31.5733,Z 73,A -154.608,B 24.8872,C -2.452,E1 24.8631,E2 -121.4004} C_DIS
LIN {X -52.1446,Y -29.184,Z 73,A -157.0966,B 24.8862,C -2.462,E1 24.8596,E2 -118.9229} C_DIS
LIN {X -53.3782,Y -26.8636,Z 73,A -159.8278,B 24.886,C -2.465,E1 24.8561,E2 -116.1843} C_DIS
LIN {X -54.6302,Y -24.2163,Z 73,A -162.6549,B 24.8853,C -2.4725,E1 24.8528,E2 -113.3596} C_DIS
LIN {X -55.7542,Y -21.5025,Z 73,A -165.5101,B 24.8846,C -2.4799,E1 24.8499,E2 -110.5061} C_DIS
LIN {X -56.7478,Y -18.7232,Z 73,A -168.3333,B 24.8838,C -2.4882,E1 24.8473,E2 -107.6867} C_DIS
LIN {X -57.5936,Y -15.933,Z 73,A -171.15,B 24.883,C -2.4962,E1 24.8451,E2 -104.8727} C_DIS
LIN {X -58.2598,Y -13.2885,Z 73,A -173.7263,B 24.8822,C -2.5047,E1 24.8434,E2 -102.3019} C_DIS
LIN {X -58.8102,Y -10.5884,Z 73,A -176.2544,B 24.8813,C -2.5148,E1 24.8421,E2 -99.7829} C_DIS
LIN {X -59.2156,Y -8.0246,Z 73,A -178.9457,B 24.8809,C -2.519,E1 24.841,E2 -97.0854} C_DIS
LIN {X -59.5388,Y -5.0997,Z 73,A 178.2272,B 24.8801,C -2.5277,E1 24.8402,E2 -94.2623} C_DIS
LIN {X -59.7149,Y -2.2356,Z 73,A 175.4373,B 24.8793,C -2.5357,E1 24.8398,E2 -91.4746} C_DIS
LIN {X -59.7532,Y 0.6523,Z 73,A 172.7549,B 24.8783,C -2.5459,E1 24.8398,E2 -88.8005} C_DIS
LIN {X -59.6849,Y 2.9326,Z 73,A 170.4413,B 24.8779,C -2.5506,E1 24.8401,E2 -86.4843} C_DIS
LIN {X -59.4672,Y 5.8761,Z 73,A 167.5952,B 24.877,C -2.5593,E1 24.8408,E2 -83.6418} C_DIS
LIN {X -59.11,Y 8.7688,Z 73,A 164.7572,B 24.8763,C -2.5674,E1 24.8418,E2 -80.8062} C_DIS
LIN {X -58.6054,Y 11.6739,Z 73,A 161.9314,B 24.8754,C -2.5763,E1 24.8433,E2 -77.985} C_DIS
LIN {X -57.9659,Y 14.5205,Z 73,A 159.1106,B 24.8746,C -2.5846,E1 24.8451,E2 -75.1675} C_DIS
LIN {X -57.188,Y 17.3325,Z 73,A 156.283,B 24.8738,C -2.5927,E1 24.8473,E2 -72.3429} C_DIS
LIN {X -56.2624,Y 20.1352,Z 73,A 153.443,B 24.873,C -2.6012,E1 24.8498,E2 -69.507} C_DIS
LIN {X -55.2088,Y 22.8666,Z 73,A 150.5909,B 24.8722,C -2.6088,E1 24.8528,E2 -66.6573} C_DIS
LIN {X -54.0087,Y 25.5721,Z 73,A 147.7624,B 24.8714,C -2.6174,E1 24.8561,E2 -63.8338} C_DIS
LIN {X -52.6958,Y 28.1786,Z 73,A 144.9447,B 24.8706,C -2.6251,E1 24.8597,E2 -61.0195} C_DIS
LIN {X -51.2563,Y 30.7194,Z 73,A 142.1047,B 24.8699,C -2.6323,E1 24.8637,E2 -58.182} C_DIS
LIN {X -49.6138,Y 33.3059,Z 73,A 139.1546,B 24.8691,C -2.6402,E1 24.8682,E2 -55.2359} C_DIS
LIN {X -47.9484,Y 35.6622,Z 73,A 136.4073,B 24.8683,C -2.6479,E1 24.8727,E2 -52.4937} C_DIS
LIN {X -46.1848,Y 37.919,Z 73,A 133.6311,B 24.8677,C -2.6545,E1 24.8775,E2 -49.7202} C_DIS
LIN {X -44.3075,Y 40.0962,Z 73,A 130.8574,B 24.867,C -2.6611,E1 24.8826,E2 -46.9497} C_DIS
LIN {X -42.2161,Y 42.2925,Z 73,A 127.9611,B 24.8663,C -2.6683,E1 24.8883,E2 -44.0581} C_DIS
LIN {X -40.0848,Y 44.3177,Z 73,A 125.1176,B 24.8657,C -2.6743,E1 24.8941,E2 -41.2175} C_DIS
LIN {X -37.9683,Y 46.1438,Z 73,A 122.401,B 24.8652,C -2.6795,E1 24.8999,E2 -38.5028} C_DIS
LIN {X -35.9024,Y 47.768,Z 73,A 120.0538,B 24.8643,C -2.6879,E1 24.905,E2 -36.167} C_DIS
LIN {X -33.7875,Y 49.2877,Z 73,A 117.3604,B 24.8642,C -2.6892,E1 24.9112,E2 -33.4676} C_DIS
LIN {X -31.3426,Y 50.8776,Z 73,A 114.5507,B 24.8637,C -2.6941,E1 24.9178,E2 -30.6607} C_DIS
LIN {X -28.8219,Y 52.3468,Z 73,A 111.7261,B 24.8633,C -2.6984,E1 24.9247,E2 -27.8381} C_DIS
LIN {X -26.2015,Y 53.7063,Z 73,A 108.8986,B 24.8628,C -2.703,E1 24.9317,E2 -25.0139} C_DIS
LIN {X -23.5406,Y 54.9248,Z 73,A 106.1612,B 24.8622,C -2.7084,E1 24.9387,E2 -22.2828} C_DIS
LIN {X -21.0235,Y 55.9356,Z 73,A 103.4833,B 24.862,C -2.7104,E1 24.9457,E2 -19.604} C_DIS
LIN {X -18.3034,Y 56.8837,Z 73,A 100.7086,B 24.8617,C -2.7134,E1 24.953,E2 -16.8313} C_DIS
LIN {X -15.6307,Y 57.6753,Z 73,A 98.0291,B 24.8615,C -2.7161,E1 24.9602,E2 -14.1539} C_DIS
LIN {X -13.0234,Y 58.3201,Z 73,A 95.461,B 24.8612,C -2.7186,E1 24.9672,E2 -11.5882} C_DIS
LIN {X -10.196,Y 58.8805,Z 73,A 92.6851,B 24.861,C -2.7204,E1 24.9748,E2 -8.8138} C_DIS
LIN {X -7.2594,Y 59.314,Z 73,A 89.837,B 24.8608,C -2.7222,E1 24.9827,E2 -5.9677} C_DIS
LIN {X -4.3787,Y 59.5962,Z 73,A 87.055,B 24.8608,C -2.7233,E1 24.9904,E2 -3.1871} C_DIS
LIN {X -1.4797,Y 59.7385,Z 73,A 84.2631,B 24.8606,C -2.724,E1 24.9982,E2 -0.3963} C_DIS
LIN {X 1.417,Y 59.7398,Z 73,A 81.4878,B 24.8606,C -2.7245,E1 25.0059,E2 2.3776} C_DIS
LIN {X 3.6091,Y 59.6475,Z 73,A 79.3669,B 24.8606,C -2.7242,E1 25.0119,E2 4.4984} C_DIS
LIN {X 6.5638,Y 59.3952,Z 73,A 76.5689,B 24.8606,C -2.7248,E1 25.0196,E2 7.2932} C_DIS
LIN {X 9.2746,Y 59.0319,Z 73,A 73.9053,B 24.8607,C -2.7233,E1 25.027,E2 9.958} C_DIS
LIN {X 12.135,Y 58.5108,Z 73,A 71.1885,B 24.8607,C -2.7236,E1 25.0344,E2 12.6708} C_DIS
LIN {X 14.8284,Y 57.8868,Z 73,A 68.6789,B 24.8605,C -2.7251,E1 25.0412,E2 15.1732} C_DIS
LIN {X 17.3574,Y 57.1804,Z 73,A 65.9691,B 24.8611,C -2.7193,E1 25.0485,E2 17.8923} C_DIS
LIN {X 20.1328,Y 56.2633,Z 73,A 63.1644,B 24.8614,C -2.7169,E1 25.0559,E2 20.6971} C_DIS
LIN {X 22.8719,Y 55.2066,Z 73,A 60.361,B 24.8616,C -2.7143,E1 25.0632,E2 23.5002} C_DIS
LIN {X 25.5483,Y 54.0201,Z 73,A 57.5596,B 24.8619,C -2.7113,E1 25.0703,E2 26.3019} C_DIS
LIN {X 28.1634,Y 52.704,Z 73,A 54.756,B 24.8623,C -2.7078,E1 25.0772,E2 29.106} C_DIS
LIN {X 30.7307,Y 51.2494,Z 73,A 51.9429,B 24.8627,C -2.7041,E1 25.084,E2 31.9192} C_DIS
LIN {X 33.2001,Y 49.6854,Z 73,A 49.1479,B 24.8631,C -2.6999,E1 25.0906,E2 34.715} C_DIS
LIN {X 35.5989,Y 47.9959,Z 73,A 46.321,B 24.8636,C -2.6949,E1 25.097,E2 37.544} C_DIS
LIN {X 37.9294,Y 46.1761,Z 73,A 43.5257,B 24.864,C -2.6906,E1 25.1031,E2 40.3388} C_DIS
LIN {X 40.1374,Y 44.2704,Z 73,A 40.7403,B 24.8646,C -2.6854,E1 25.1089,E2 43.1255} C_DIS
LIN {X 42.2512,Y 42.2578,Z 73,A 37.9513,B 24.8651,C -2.6799,E1 25.1145,E2 45.916} C_DIS
LIN {X 44.28,Y 40.1269,Z 73,A 35.1437,B 24.8657,C -2.674,E1 25.1198,E2 48.725} C_DIS
LIN {X 46.1926,Y 37.9095,Z 73,A 32.3423,B 24.8664,C -2.6678,E1 25.1249,E2 51.5284} C_DIS
Enddeposition()
END
